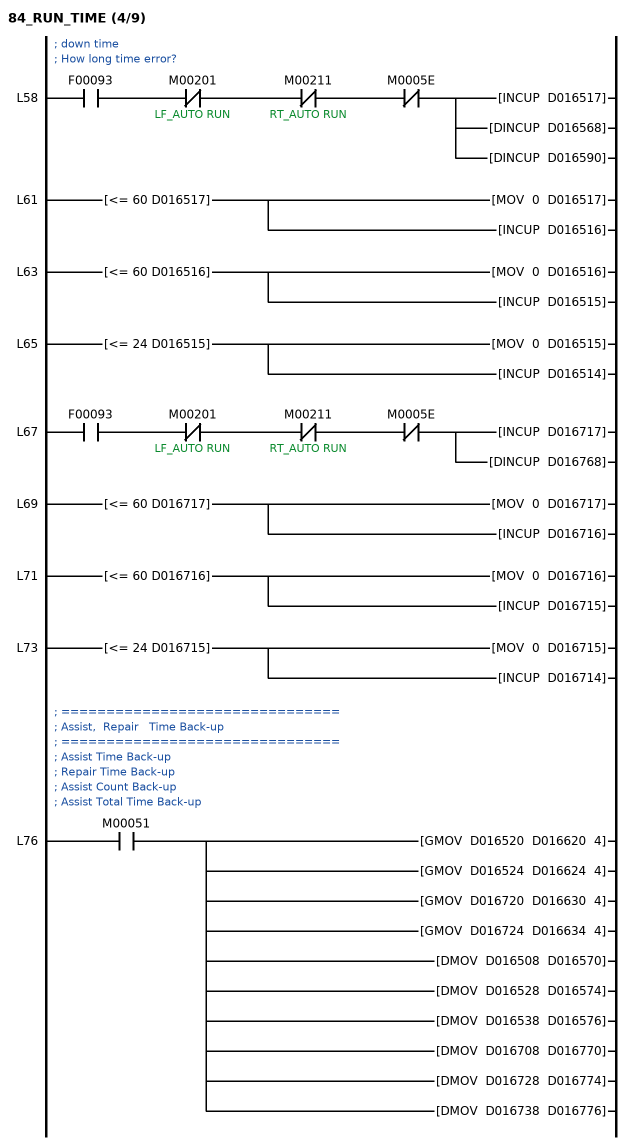
[picture p360: 84_RUN_TIME rungs L58-L76]
; L58
LOAD      F00093
AND NOT   M00201	// LF_AUTO RUN
AND NOT   M00211	// RT_AUTO RUN
AND NOT   M0005E
INCUP     D016517
DINCUP    D016568
DINCUP    D016590
// output comment: down time
// output comment: How long time error?
; L61
LOAD<=    60 D016517
MOV       0 D016517
INCUP     D016516
; L63
LOAD<=    60 D016516
MOV       0 D016516
INCUP     D016515
; L65
LOAD<=    24 D016515
MOV       0 D016515
INCUP     D016514
; L67
LOAD      F00093
AND NOT   M00201	// LF_AUTO RUN
AND NOT   M00211	// RT_AUTO RUN
AND NOT   M0005E
INCUP     D016717
DINCUP    D016768
; L69
LOAD<=    60 D016717
MOV       0 D016717
INCUP     D016716
; L71
LOAD<=    60 D016716
MOV       0 D016716
INCUP     D016715
; L73
LOAD<=    24 D016715
MOV       0 D016715
INCUP     D016714
// ===============================
// Assist,  Repair   Time Back-up
// ===============================
; L76
LOAD      M00051
GMOV      D016520 D016620 4
GMOV      D016524 D016624 4
GMOV      D016720 D016630 4
GMOV      D016724 D016634 4
DMOV      D016508 D016570
DMOV      D016528 D016574
DMOV      D016538 D016576
DMOV      D016708 D016770
DMOV      D016728 D016774
DMOV      D016738 D016776
// output comment: Assist Time Back-up
// output comment: Repair Time Back-up
// output comment: Assist Count Back-up
// output comment: Assist Total Time Back-up

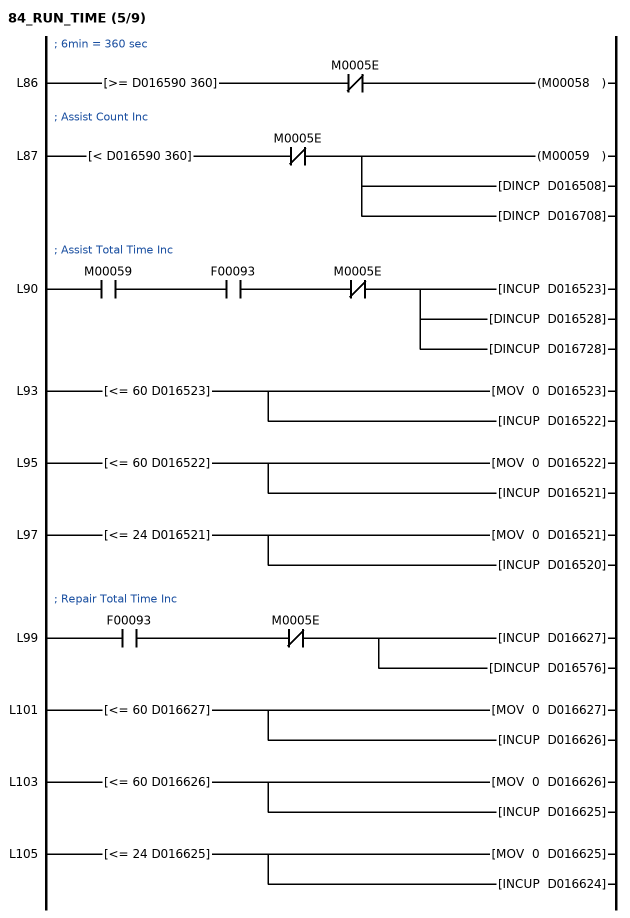
; L86
LOAD>=    D016590 360
AND NOT   M0005E
OUT       M00058
// output comment: 6min = 360 sec
; L87
LOAD<     D016590 360
AND NOT   M0005E
OUT       M00059
DINCP     D016508
DINCP     D016708
// output comment: Assist Count Inc
; L90
LOAD      M00059
AND       F00093
AND NOT   M0005E
INCUP     D016523
DINCUP    D016528
DINCUP    D016728
// output comment: Assist Total Time Inc
; L93
LOAD<=    60 D016523
MOV       0 D016523
INCUP     D016522
; L95
LOAD<=    60 D016522
MOV       0 D016522
INCUP     D016521
; L97
LOAD<=    24 D016521
MOV       0 D016521
INCUP     D016520
; L99
LOAD      F00093
AND NOT   M0005E
INCUP     D016627
DINCUP    D016576
// output comment: Repair Total Time Inc
; L101
LOAD<=    60 D016627
MOV       0 D016627
INCUP     D016626
; L103
LOAD<=    60 D016626
MOV       0 D016626
INCUP     D016625
; L105
LOAD<=    24 D016625
MOV       0 D016625
INCUP     D016624

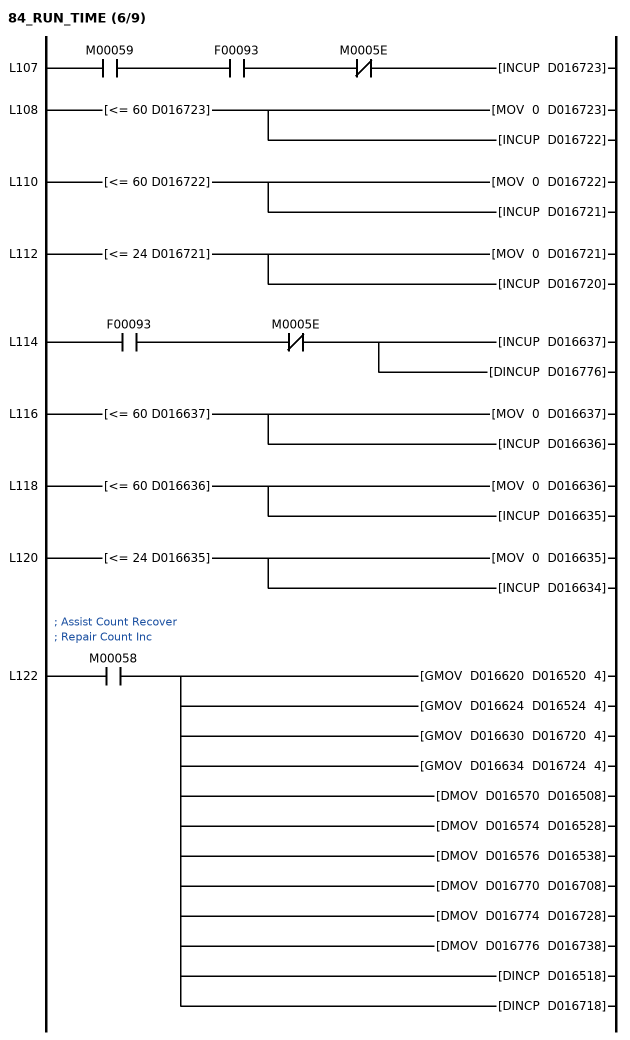
; L107
LOAD      M00059
AND       F00093
AND NOT   M0005E
INCUP     D016723
; L108
LOAD<=    60 D016723
MOV       0 D016723
INCUP     D016722
; L110
LOAD<=    60 D016722
MOV       0 D016722
INCUP     D016721
; L112
LOAD<=    24 D016721
MOV       0 D016721
INCUP     D016720
; L114
LOAD      F00093
AND NOT   M0005E
INCUP     D016637
DINCUP    D016776
; L116
LOAD<=    60 D016637
MOV       0 D016637
INCUP     D016636
; L118
LOAD<=    60 D016636
MOV       0 D016636
INCUP     D016635
; L120
LOAD<=    24 D016635
MOV       0 D016635
INCUP     D016634
; L122
LOAD      M00058
GMOV      D016620 D016520 4
GMOV      D016624 D016524 4
GMOV      D016630 D016720 4
GMOV      D016634 D016724 4
DMOV      D016570 D016508
DMOV      D016574 D016528
DMOV      D016576 D016538
DMOV      D016770 D016708
DMOV      D016774 D016728
DMOV      D016776 D016738
DINCP     D016518
DINCP     D016718
// output comment: Assist Count Recover
// output comment: Repair Count Inc

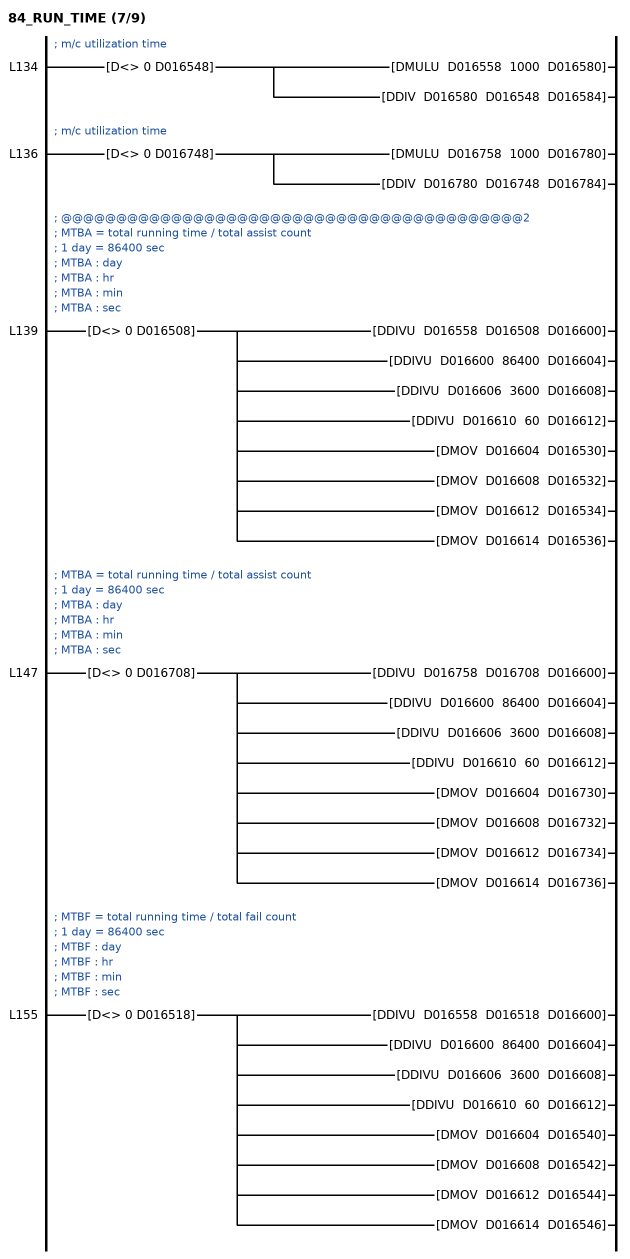
; L134
LOADD<>   0 D016548
DMULU     D016558 1000 D016580
DDIV      D016580 D016548 D016584
// output comment: m/c utilization time
; L136
LOADD<>   0 D016748
DMULU     D016758 1000 D016780
DDIV      D016780 D016748 D016784
// output comment: m/c utilization time
// @@@@@@@@@@@@@@@@@@@@@@@@@@@@@@@@@@@@@@@@@@2
; L139
LOADD<>   0 D016508
DDIVU     D016558 D016508 D016600
DDIVU     D016600 86400 D016604
DDIVU     D016606 3600 D016608
DDIVU     D016610 60 D016612
DMOV      D016604 D016530
DMOV      D016608 D016532
DMOV      D016612 D016534
DMOV      D016614 D016536
// output comment: MTBA = total running time / total assist count
// output comment: 1 day = 86400 sec
// output comment: MTBA : day
// output comment: MTBA : hr
// output comment: MTBA : min
// output comment: MTBA : sec
; L147
LOADD<>   0 D016708
DDIVU     D016758 D016708 D016600
DDIVU     D016600 86400 D016604
DDIVU     D016606 3600 D016608
DDIVU     D016610 60 D016612
DMOV      D016604 D016730
DMOV      D016608 D016732
DMOV      D016612 D016734
DMOV      D016614 D016736
// output comment: MTBA = total running time / total assist count
// output comment: 1 day = 86400 sec
// output comment: MTBA : day
// output comment: MTBA : hr
// output comment: MTBA : min
// output comment: MTBA : sec
; L155
LOADD<>   0 D016518
DDIVU     D016558 D016518 D016600
DDIVU     D016600 86400 D016604
DDIVU     D016606 3600 D016608
DDIVU     D016610 60 D016612
DMOV      D016604 D016540
DMOV      D016608 D016542
DMOV      D016612 D016544
DMOV      D016614 D016546
// output comment: MTBF = total running time / total fail count
// output comment: 1 day = 86400 sec
// output comment: MTBF : day
// output comment: MTBF : hr
// output comment: MTBF : min
// output comment: MTBF : sec

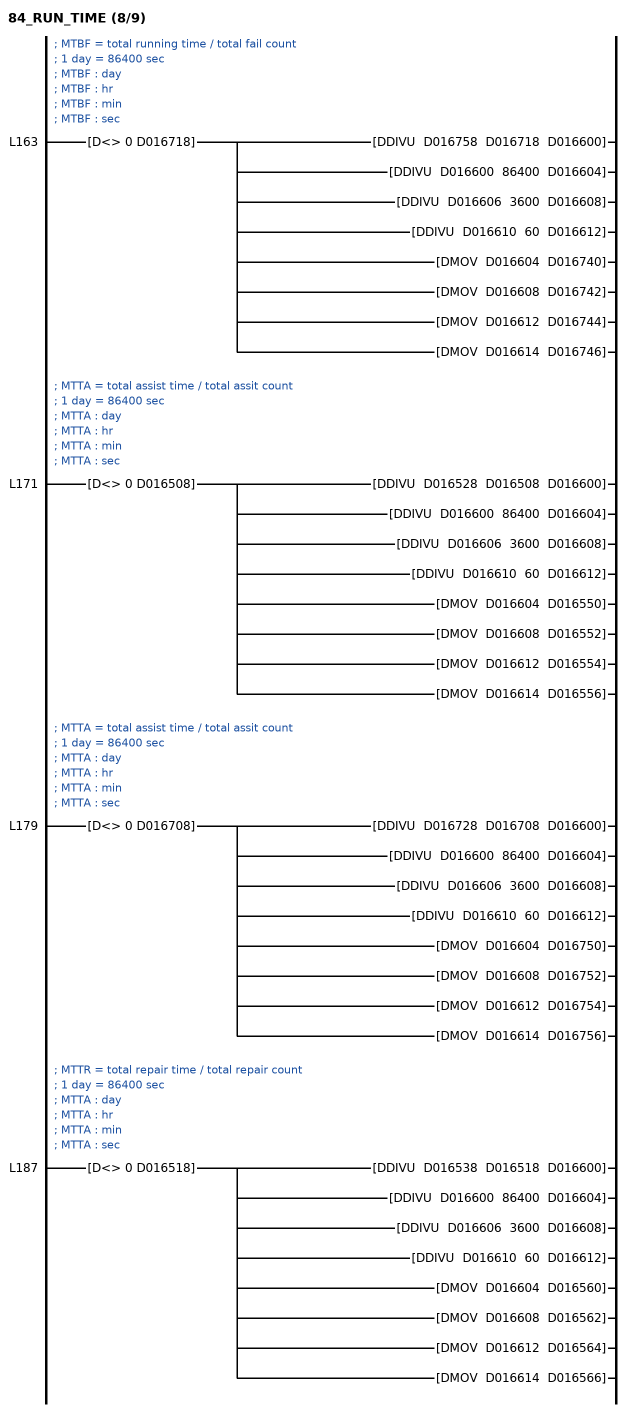
; L163
LOADD<>   0 D016718
DDIVU     D016758 D016718 D016600
DDIVU     D016600 86400 D016604
DDIVU     D016606 3600 D016608
DDIVU     D016610 60 D016612
DMOV      D016604 D016740
DMOV      D016608 D016742
DMOV      D016612 D016744
DMOV      D016614 D016746
// output comment: MTBF = total running time / total fail count
// output comment: 1 day = 86400 sec
// output comment: MTBF : day
// output comment: MTBF : hr
// output comment: MTBF : min
// output comment: MTBF : sec
; L171
LOADD<>   0 D016508
DDIVU     D016528 D016508 D016600
DDIVU     D016600 86400 D016604
DDIVU     D016606 3600 D016608
DDIVU     D016610 60 D016612
DMOV      D016604 D016550
DMOV      D016608 D016552
DMOV      D016612 D016554
DMOV      D016614 D016556
// output comment: MTTA = total assist time / total assit count
// output comment: 1 day = 86400 sec
// output comment: MTTA : day
// output comment: MTTA : hr
// output comment: MTTA : min
// output comment: MTTA : sec
; L179
LOADD<>   0 D016708
DDIVU     D016728 D016708 D016600
DDIVU     D016600 86400 D016604
DDIVU     D016606 3600 D016608
DDIVU     D016610 60 D016612
DMOV      D016604 D016750
DMOV      D016608 D016752
DMOV      D016612 D016754
DMOV      D016614 D016756
// output comment: MTTA = total assist time / total assit count
// output comment: 1 day = 86400 sec
// output comment: MTTA : day
// output comment: MTTA : hr
// output comment: MTTA : min
// output comment: MTTA : sec
; L187
LOADD<>   0 D016518
DDIVU     D016538 D016518 D016600
DDIVU     D016600 86400 D016604
DDIVU     D016606 3600 D016608
DDIVU     D016610 60 D016612
DMOV      D016604 D016560
DMOV      D016608 D016562
DMOV      D016612 D016564
DMOV      D016614 D016566
// output comment: MTTR = total repair time / total repair count
// output comment: 1 day = 86400 sec
// output comment: MTTA : day
// output comment: MTTA : hr
// output comment: MTTA : min
// output comment: MTTA : sec

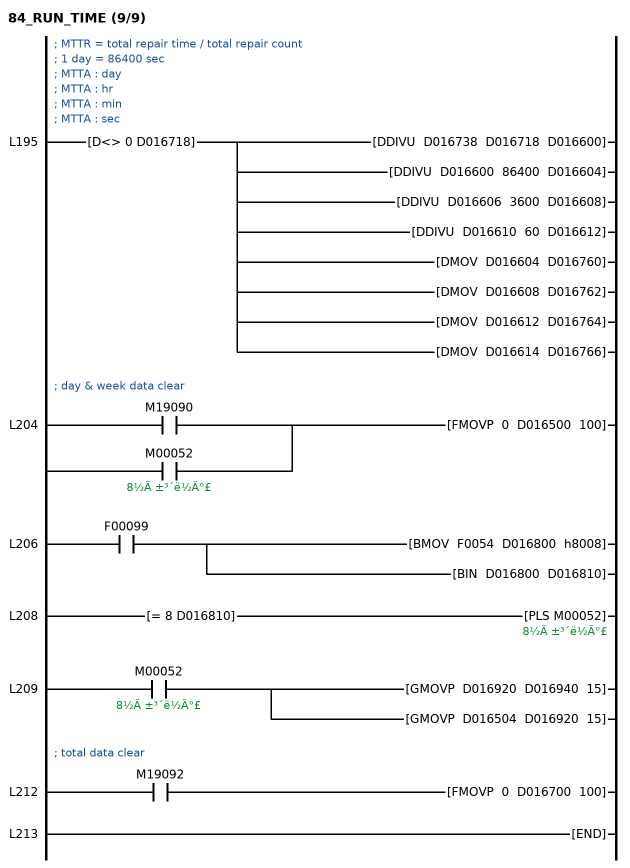
; L195
LOADD<>   0 D016718
DDIVU     D016738 D016718 D016600
DDIVU     D016600 86400 D016604
DDIVU     D016606 3600 D016608
DDIVU     D016610 60 D016612
DMOV      D016604 D016760
DMOV      D016608 D016762
DMOV      D016612 D016764
DMOV      D016614 D016766
// output comment: MTTR = total repair time / total repair count
// output comment: 1 day = 86400 sec
// output comment: MTTA : day
// output comment: MTTA : hr
// output comment: MTTA : min
// output comment: MTTA : sec
// day & week data clear
; L204
LOAD      M19090
OR        M00052	// 8½Ã ±³´ë½Ã°£
FMOVP     0 D016500 100
; L206
LOAD      F00099
BMOV      F0054 D016800 h8008
BIN       D016800 D016810
; L208
LOAD=     8 D016810
OUTP      M00052	// 8½Ã ±³´ë½Ã°£
; L209
LOAD      M00052	// 8½Ã ±³´ë½Ã°£
GMOVP     D016920 D016940 15
GMOVP     D016504 D016920 15
// total data clear
; L212
LOAD      M19092
FMOVP     0 D016700 100
; L213
END

PROGRAM 90_ALARM (task: ½ºÄµ ÇÁ·Î±×·¥)

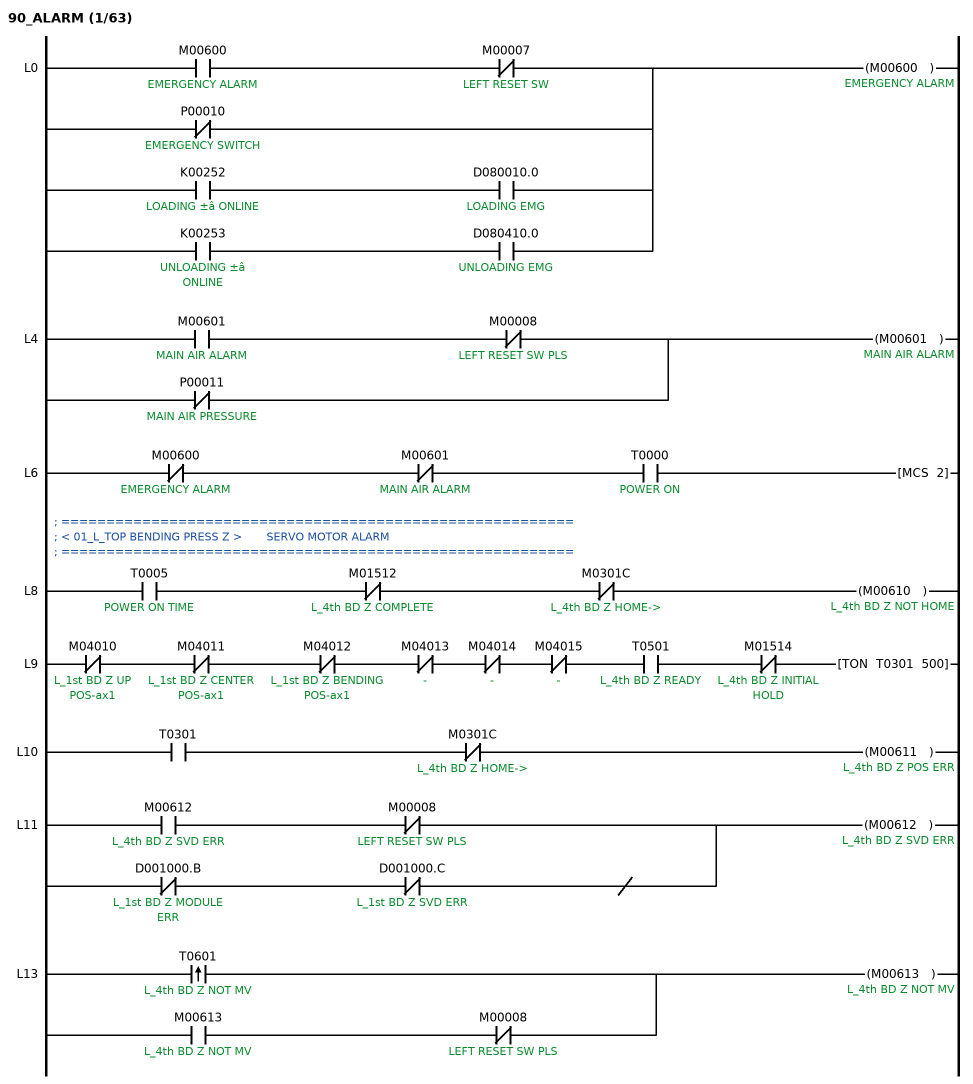
; L0
LOAD      M00600	// EMERGENCY ALARM
AND NOT   M00007	// LEFT RESET SW
OR NOT    P00010	// EMERGENCY SWITCH
LOAD      K00252	// LOADING ±â ONLINE
AND       D080010.0	// LOADING EMG
OR LOAD
LOAD      K00253	// UNLOADING ±â ONLINE
AND       D080410.0	// UNLOADING EMG
OR LOAD
OUT       M00600	// EMERGENCY ALARM
; L4
LOAD      M00601	// MAIN AIR ALARM
AND NOT   M00008	// LEFT RESET SW PLS
OR NOT    P00011	// MAIN AIR PRESSURE
OUT       M00601	// MAIN AIR ALARM
; L6
LOAD NOT  M00600	// EMERGENCY ALARM
AND NOT   M00601	// MAIN AIR ALARM
AND       T0000	// POWER ON
MCS       2
// =========================================================
// 
//        < 01_L_TOP BENDING PRESS Z >       SERVO MOTOR ALARM
// 
// =========================================================
; L8
LOAD      T0005	// POWER ON TIME
AND NOT   M01512	// L_4th BD Z COMPLETE
AND NOT   M0301C	// L_4th BD Z HOME->
OUT       M00610	// L_4th BD Z NOT HOME
; L9
LOAD NOT  M04010	// L_1st BD Z UP POS-ax1
AND NOT   M04011	// L_1st BD Z CENTER POS-ax1
AND NOT   M04012	// L_1st BD Z BENDING POS-ax1
AND NOT   M04013	// -
AND NOT   M04014	// -
AND NOT   M04015	// -
AND       T0501	// L_4th BD Z READY
AND NOT   M01514	// L_4th BD Z INITIAL HOLD
TON       T0301 500
; L10
LOAD      T0301
AND NOT   M0301C	// L_4th BD Z HOME->
OUT       M00611	// L_4th BD Z POS ERR
; L11
LOAD      M00612	// L_4th BD Z SVD ERR
AND NOT   M00008	// LEFT RESET SW PLS
LOAD NOT  D001000.B	// L_1st BD Z MODULE ERR
AND NOT   D001000.C	// L_1st BD Z SVD ERR
NOT
OR LOAD
OUT       M00612	// L_4th BD Z SVD ERR
; L13
LOADP     T0601	// L_4th BD Z NOT MV
LOAD      M00613	// L_4th BD Z NOT MV
AND NOT   M00008	// LEFT RESET SW PLS
OR LOAD
OUT       M00613	// L_4th BD Z NOT MV

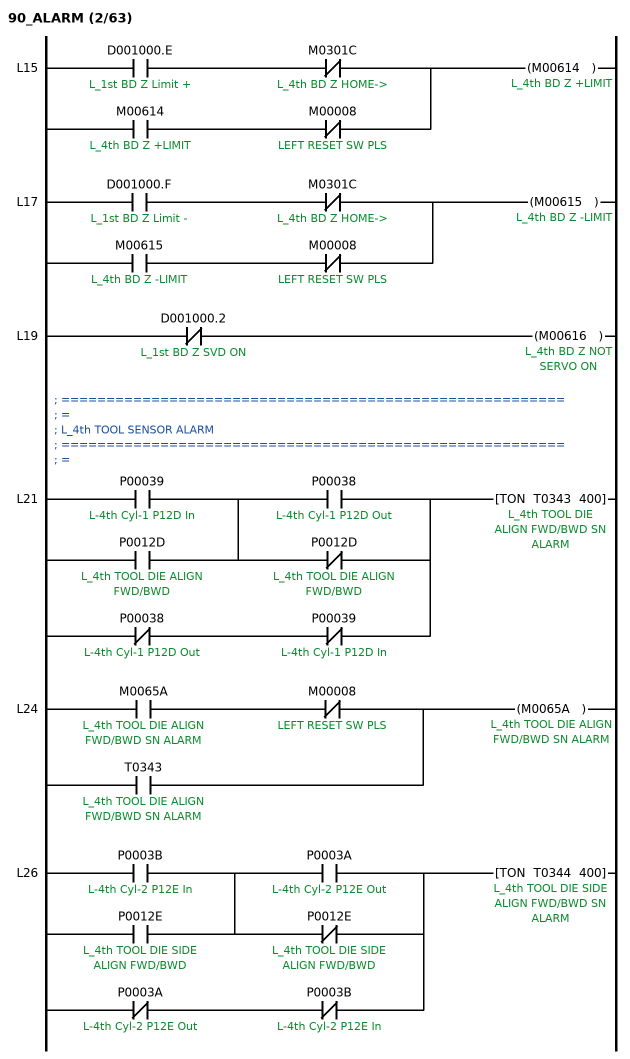
; L15
LOAD      D001000.E	// L_1st BD Z Limit +
AND NOT   M0301C	// L_4th BD Z HOME->
LOAD      M00614	// L_4th BD Z +LIMIT
AND NOT   M00008	// LEFT RESET SW PLS
OR LOAD
OUT       M00614	// L_4th BD Z +LIMIT
; L17
LOAD      D001000.F	// L_1st BD Z Limit -
AND NOT   M0301C	// L_4th BD Z HOME->
LOAD      M00615	// L_4th BD Z -LIMIT
AND NOT   M00008	// LEFT RESET SW PLS
OR LOAD
OUT       M00615	// L_4th BD Z -LIMIT
; L19
LOAD NOT  D001000.2	// L_1st BD Z SVD ON
OUT       M00616	// L_4th BD Z NOT SERVO ON
// =========================================================
// 
//        L_4th TOOL SENSOR ALARM
// 
// =========================================================
; L21
LOAD      P00039	// L-4th Cyl-1 P12D In
OR        P0012D	// L_4th TOOL DIE ALIGN FWD/BWD
LOAD      P00038	// L-4th Cyl-1 P12D Out
OR NOT    P0012D	// L_4th TOOL DIE ALIGN FWD/BWD
AND LOAD
LOAD NOT  P00038	// L-4th Cyl-1 P12D Out
AND NOT   P00039	// L-4th Cyl-1 P12D In
OR LOAD
TON       T0343 400	// L_4th TOOL DIE ALIGN FWD/BWD SN ALARM
; L24
LOAD      M0065A	// L_4th TOOL DIE ALIGN FWD/BWD SN ALARM
AND NOT   M00008	// LEFT RESET SW PLS
OR        T0343	// L_4th TOOL DIE ALIGN FWD/BWD SN ALARM
OUT       M0065A	// L_4th TOOL DIE ALIGN FWD/BWD SN ALARM
; L26
LOAD      P0003B	// L-4th Cyl-2 P12E In
OR        P0012E	// L_4th TOOL DIE SIDE ALIGN FWD/BWD
LOAD      P0003A	// L-4th Cyl-2 P12E Out
OR NOT    P0012E	// L_4th TOOL DIE SIDE ALIGN FWD/BWD
AND LOAD
LOAD NOT  P0003A	// L-4th Cyl-2 P12E Out
AND NOT   P0003B	// L-4th Cyl-2 P12E In
OR LOAD
TON       T0344 400	// L_4th TOOL DIE SIDE ALIGN FWD/BWD SN ALARM

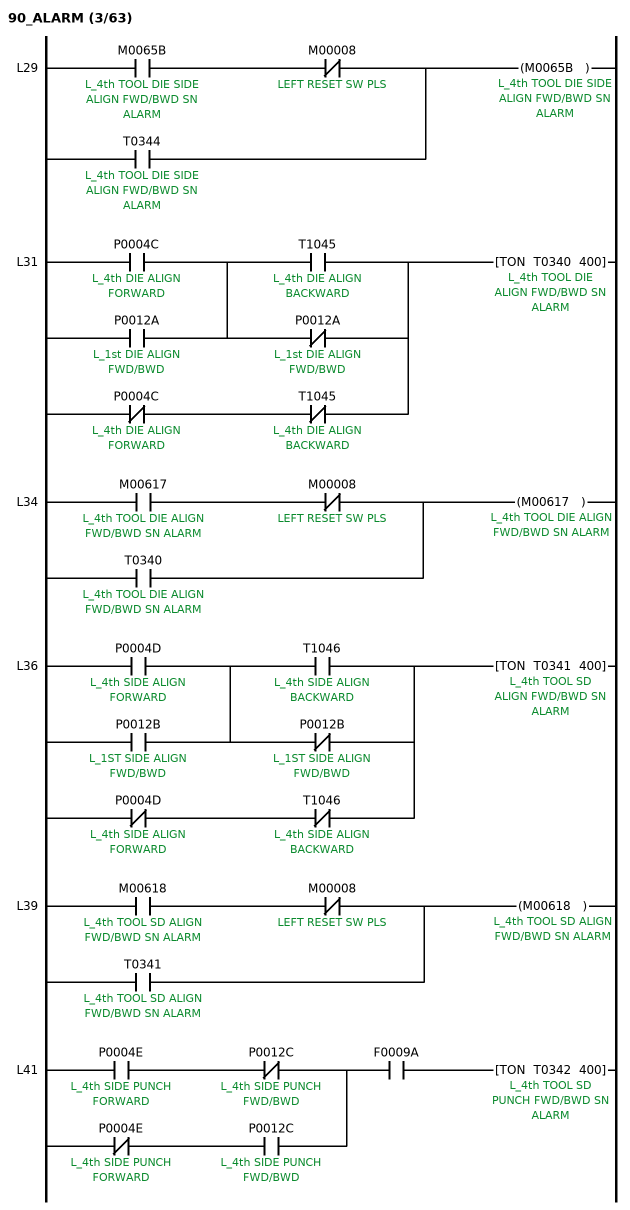
; L29
LOAD      M0065B	// L_4th TOOL DIE SIDE ALIGN FWD/BWD SN ALARM
AND NOT   M00008	// LEFT RESET SW PLS
OR        T0344	// L_4th TOOL DIE SIDE ALIGN FWD/BWD SN ALARM
OUT       M0065B	// L_4th TOOL DIE SIDE ALIGN FWD/BWD SN ALARM
; L31
LOAD      P0004C	// L_4th DIE ALIGN FORWARD
OR        P0012A	// L_1st DIE ALIGN FWD/BWD
LOAD      T1045	// L_4th DIE ALIGN BACKWARD
OR NOT    P0012A	// L_1st DIE ALIGN FWD/BWD
AND LOAD
LOAD NOT  P0004C	// L_4th DIE ALIGN FORWARD
AND NOT   T1045	// L_4th DIE ALIGN BACKWARD
OR LOAD
TON       T0340 400	// L_4th TOOL DIE ALIGN FWD/BWD SN ALARM
; L34
LOAD      M00617	// L_4th TOOL DIE ALIGN FWD/BWD SN ALARM
AND NOT   M00008	// LEFT RESET SW PLS
OR        T0340	// L_4th TOOL DIE ALIGN FWD/BWD SN ALARM
OUT       M00617	// L_4th TOOL DIE ALIGN FWD/BWD SN ALARM
; L36
LOAD      P0004D	// L_4th SIDE ALIGN FORWARD
OR        P0012B	// L_1ST SIDE ALIGN FWD/BWD
LOAD      T1046	// L_4th SIDE ALIGN BACKWARD
OR NOT    P0012B	// L_1ST SIDE ALIGN FWD/BWD
AND LOAD
LOAD NOT  P0004D	// L_4th SIDE ALIGN FORWARD
AND NOT   T1046	// L_4th SIDE ALIGN BACKWARD
OR LOAD
TON       T0341 400	// L_4th TOOL SD ALIGN FWD/BWD SN ALARM
; L39
LOAD      M00618	// L_4th TOOL SD ALIGN FWD/BWD SN ALARM
AND NOT   M00008	// LEFT RESET SW PLS
OR        T0341	// L_4th TOOL SD ALIGN FWD/BWD SN ALARM
OUT       M00618	// L_4th TOOL SD ALIGN FWD/BWD SN ALARM
; L41
LOAD      P0004E	// L_4th SIDE PUNCH FORWARD
AND NOT   P0012C	// L_4th SIDE PUNCH FWD/BWD
LOAD NOT  P0004E	// L_4th SIDE PUNCH FORWARD
AND       P0012C	// L_4th SIDE PUNCH FWD/BWD
OR LOAD
AND       F0009A
TON       T0342 400	// L_4th TOOL SD PUNCH FWD/BWD SN ALARM

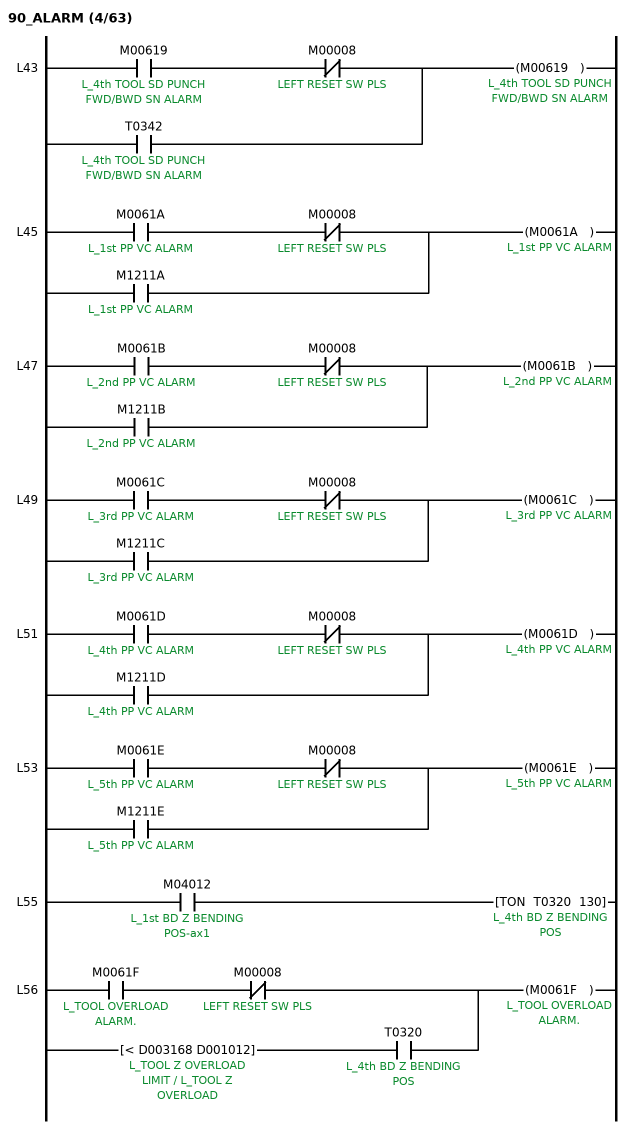
; L43
LOAD      M00619	// L_4th TOOL SD PUNCH FWD/BWD SN ALARM
AND NOT   M00008	// LEFT RESET SW PLS
OR        T0342	// L_4th TOOL SD PUNCH FWD/BWD SN ALARM
OUT       M00619	// L_4th TOOL SD PUNCH FWD/BWD SN ALARM
; L45
LOAD      M0061A	// L_1st PP VC ALARM
AND NOT   M00008	// LEFT RESET SW PLS
OR        M1211A	// L_1st PP VC ALARM
OUT       M0061A	// L_1st PP VC ALARM
; L47
LOAD      M0061B	// L_2nd PP VC ALARM
AND NOT   M00008	// LEFT RESET SW PLS
OR        M1211B	// L_2nd PP VC ALARM
OUT       M0061B	// L_2nd PP VC ALARM
; L49
LOAD      M0061C	// L_3rd PP VC ALARM
AND NOT   M00008	// LEFT RESET SW PLS
OR        M1211C	// L_3rd PP VC ALARM
OUT       M0061C	// L_3rd PP VC ALARM
; L51
LOAD      M0061D	// L_4th PP VC ALARM
AND NOT   M00008	// LEFT RESET SW PLS
OR        M1211D	// L_4th PP VC ALARM
OUT       M0061D	// L_4th PP VC ALARM
; L53
LOAD      M0061E	// L_5th PP VC ALARM
AND NOT   M00008	// LEFT RESET SW PLS
OR        M1211E	// L_5th PP VC ALARM
OUT       M0061E	// L_5th PP VC ALARM
; L55
LOAD      M04012	// L_1st BD Z BENDING POS-ax1
TON       T0320 130	// L_4th BD Z BENDING POS
; L56
LOAD      M0061F	// L_TOOL OVERLOAD ALARM.
AND NOT   M00008	// LEFT RESET SW PLS
LOAD<     D003168 D001012	// L_TOOL Z OVERLOAD LIMIT / L_TOOL Z OVERLOAD
AND       T0320	// L_4th BD Z BENDING POS
OR LOAD
OUT       M0061F	// L_TOOL OVERLOAD ALARM.

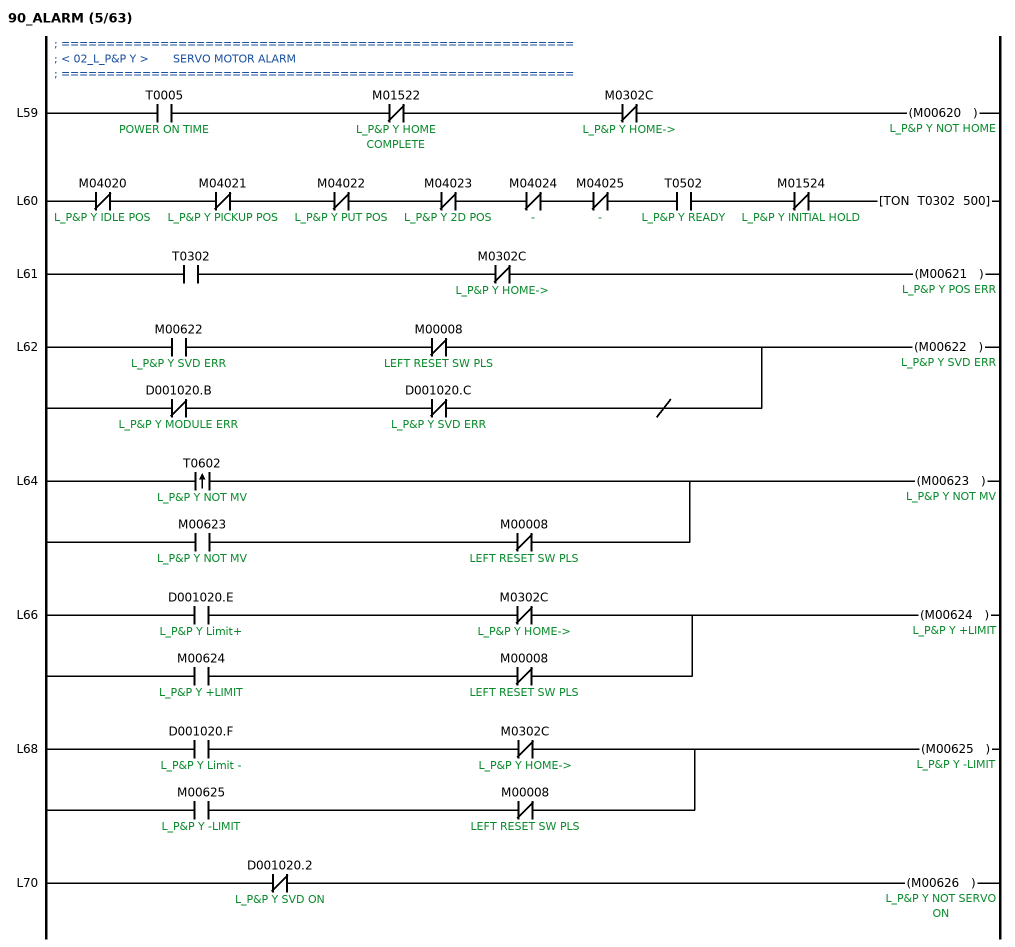
// =========================================================
// 
//        < 02_L_P&P Y >       SERVO MOTOR ALARM
// 
// =========================================================
; L59
LOAD      T0005	// POWER ON TIME
AND NOT   M01522	// L_P&P Y HOME COMPLETE
AND NOT   M0302C	// L_P&P Y HOME->
OUT       M00620	// L_P&P Y NOT HOME
; L60
LOAD NOT  M04020	// L_P&P Y IDLE POS
AND NOT   M04021	// L_P&P Y PICKUP POS
AND NOT   M04022	// L_P&P Y PUT POS
AND NOT   M04023	// L_P&P Y 2D POS
AND NOT   M04024	// -
AND NOT   M04025	// -
AND       T0502	// L_P&P Y READY
AND NOT   M01524	// L_P&P Y INITIAL HOLD
TON       T0302 500
; L61
LOAD      T0302
AND NOT   M0302C	// L_P&P Y HOME->
OUT       M00621	// L_P&P Y POS ERR
; L62
LOAD      M00622	// L_P&P Y SVD ERR
AND NOT   M00008	// LEFT RESET SW PLS
LOAD NOT  D001020.B	// L_P&P Y MODULE ERR
AND NOT   D001020.C	// L_P&P Y SVD ERR
NOT
OR LOAD
OUT       M00622	// L_P&P Y SVD ERR
; L64
LOADP     T0602	// L_P&P Y NOT MV
LOAD      M00623	// L_P&P Y NOT MV
AND NOT   M00008	// LEFT RESET SW PLS
OR LOAD
OUT       M00623	// L_P&P Y NOT MV
; L66
LOAD      D001020.E	// L_P&P Y Limit+
AND NOT   M0302C	// L_P&P Y HOME->
LOAD      M00624	// L_P&P Y +LIMIT
AND NOT   M00008	// LEFT RESET SW PLS
OR LOAD
OUT       M00624	// L_P&P Y +LIMIT
; L68
LOAD      D001020.F	// L_P&P Y Limit -
AND NOT   M0302C	// L_P&P Y HOME->
LOAD      M00625	// L_P&P Y -LIMIT
AND NOT   M00008	// LEFT RESET SW PLS
OR LOAD
OUT       M00625	// L_P&P Y -LIMIT
; L70
LOAD NOT  D001020.2	// L_P&P Y SVD ON
OUT       M00626	// L_P&P Y NOT SERVO ON

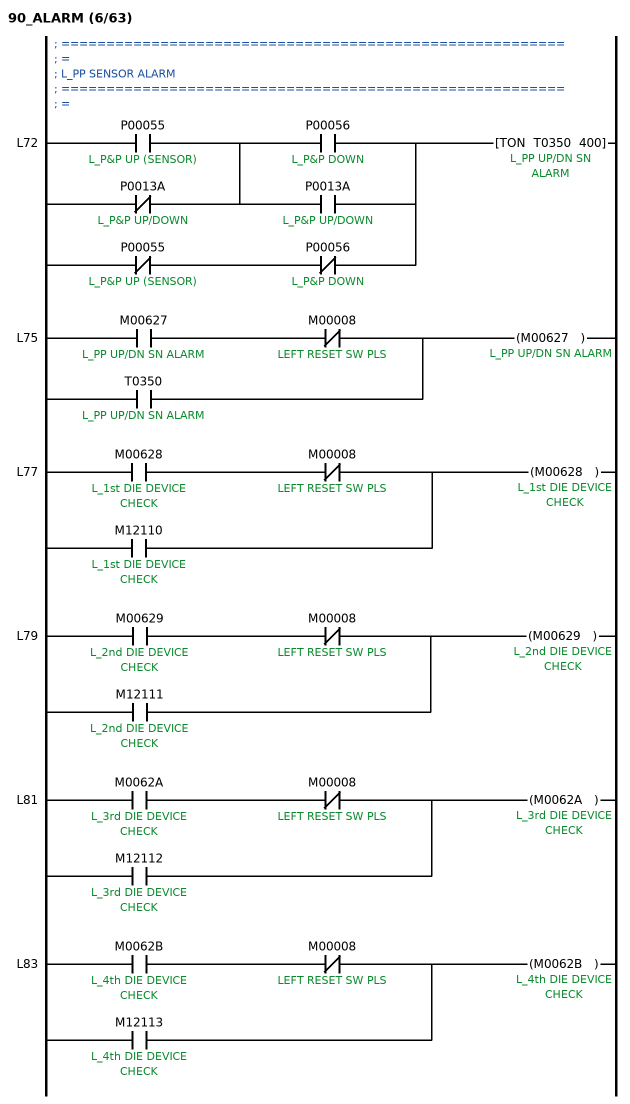
// =========================================================
// 
//       L_PP SENSOR ALARM
// 
// =========================================================
; L72
LOAD      P00055	// L_P&P UP (SENSOR)
OR NOT    P0013A	// L_P&P UP/DOWN
LOAD      P00056	// L_P&P DOWN
OR        P0013A	// L_P&P UP/DOWN
AND LOAD
LOAD NOT  P00055	// L_P&P UP (SENSOR)
AND NOT   P00056	// L_P&P DOWN
OR LOAD
TON       T0350 400	// L_PP UP/DN SN ALARM
; L75
LOAD      M00627	// L_PP UP/DN SN ALARM
AND NOT   M00008	// LEFT RESET SW PLS
OR        T0350	// L_PP UP/DN SN ALARM
OUT       M00627	// L_PP UP/DN SN ALARM
; L77
LOAD      M00628	// L_1st DIE DEVICE CHECK
AND NOT   M00008	// LEFT RESET SW PLS
OR        M12110	// L_1st DIE DEVICE CHECK
OUT       M00628	// L_1st DIE DEVICE CHECK
; L79
LOAD      M00629	// L_2nd DIE DEVICE CHECK
AND NOT   M00008	// LEFT RESET SW PLS
OR        M12111	// L_2nd DIE DEVICE CHECK
OUT       M00629	// L_2nd DIE DEVICE CHECK
; L81
LOAD      M0062A	// L_3rd DIE DEVICE CHECK
AND NOT   M00008	// LEFT RESET SW PLS
OR        M12112	// L_3rd DIE DEVICE CHECK
OUT       M0062A	// L_3rd DIE DEVICE CHECK
; L83
LOAD      M0062B	// L_4th DIE DEVICE CHECK
AND NOT   M00008	// LEFT RESET SW PLS
OR        M12113	// L_4th DIE DEVICE CHECK
OUT       M0062B	// L_4th DIE DEVICE CHECK

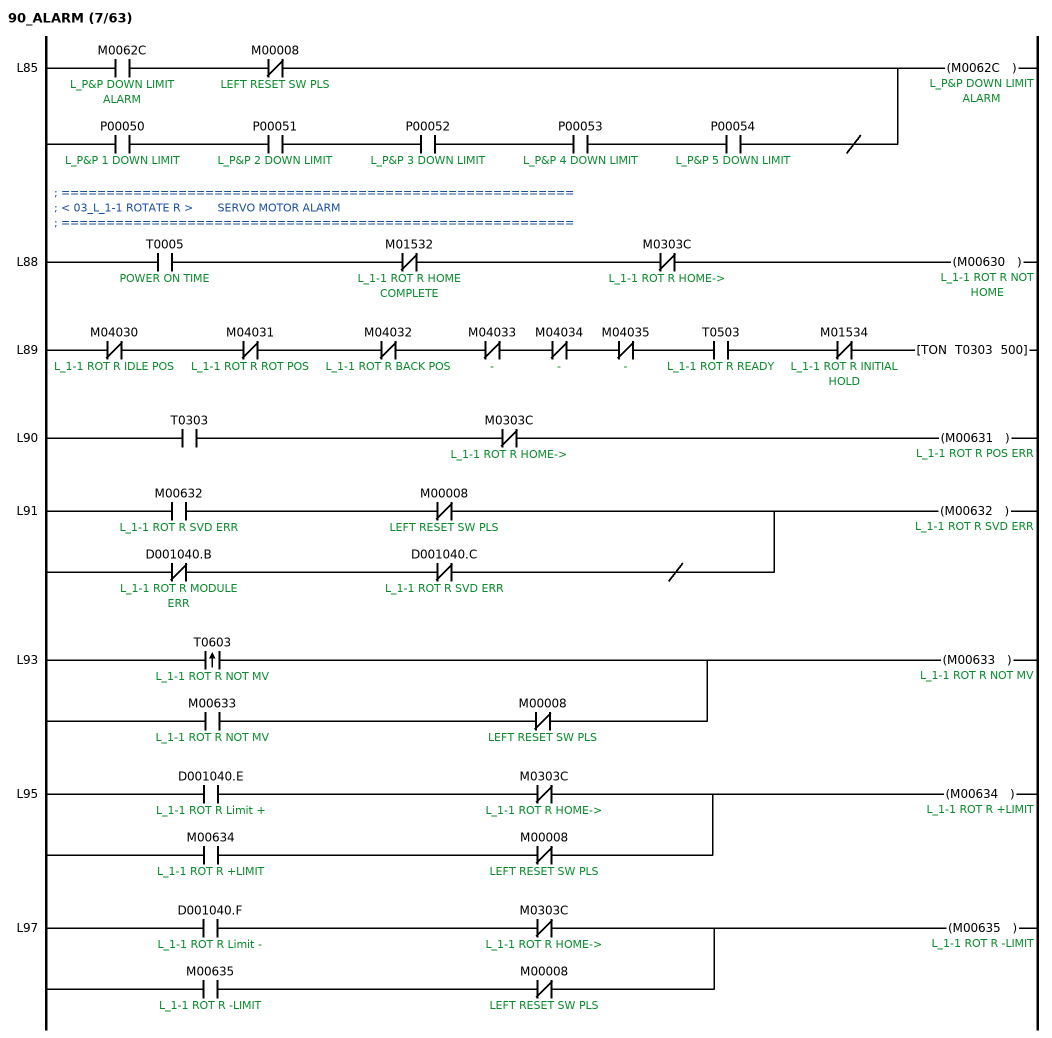
; L85
LOAD      M0062C	// L_P&P DOWN LIMIT ALARM
AND NOT   M00008	// LEFT RESET SW PLS
LOAD      P00050	// L_P&P 1 DOWN LIMIT
AND       P00051	// L_P&P 2 DOWN LIMIT
AND       P00052	// L_P&P 3 DOWN LIMIT
AND       P00053	// L_P&P 4 DOWN LIMIT
AND       P00054	// L_P&P 5 DOWN LIMIT
NOT
OR LOAD
OUT       M0062C	// L_P&P DOWN LIMIT ALARM
// =========================================================
// 
//        < 03_L_1-1 ROTATE R >       SERVO MOTOR ALARM
// 
// =========================================================
; L88
LOAD      T0005	// POWER ON TIME
AND NOT   M01532	// L_1-1 ROT R HOME COMPLETE
AND NOT   M0303C	// L_1-1 ROT R HOME->
OUT       M00630	// L_1-1 ROT R NOT HOME
; L89
LOAD NOT  M04030	// L_1-1 ROT R IDLE POS
AND NOT   M04031	// L_1-1 ROT R ROT POS
AND NOT   M04032	// L_1-1 ROT R BACK POS
AND NOT   M04033	// -
AND NOT   M04034	// -
AND NOT   M04035	// -
AND       T0503	// L_1-1 ROT R READY
AND NOT   M01534	// L_1-1 ROT R INITIAL HOLD
TON       T0303 500
; L90
LOAD      T0303
AND NOT   M0303C	// L_1-1 ROT R HOME->
OUT       M00631	// L_1-1 ROT R POS ERR
; L91
LOAD      M00632	// L_1-1 ROT R SVD ERR
AND NOT   M00008	// LEFT RESET SW PLS
LOAD NOT  D001040.B	// L_1-1 ROT R MODULE ERR
AND NOT   D001040.C	// L_1-1 ROT R SVD ERR
NOT
OR LOAD
OUT       M00632	// L_1-1 ROT R SVD ERR
; L93
LOADP     T0603	// L_1-1 ROT R NOT MV
LOAD      M00633	// L_1-1 ROT R NOT MV
AND NOT   M00008	// LEFT RESET SW PLS
OR LOAD
OUT       M00633	// L_1-1 ROT R NOT MV
; L95
LOAD      D001040.E	// L_1-1 ROT R Limit +
AND NOT   M0303C	// L_1-1 ROT R HOME->
LOAD      M00634	// L_1-1 ROT R +LIMIT
AND NOT   M00008	// LEFT RESET SW PLS
OR LOAD
OUT       M00634	// L_1-1 ROT R +LIMIT
; L97
LOAD      D001040.F	// L_1-1 ROT R Limit -
AND NOT   M0303C	// L_1-1 ROT R HOME->
LOAD      M00635	// L_1-1 ROT R -LIMIT
AND NOT   M00008	// LEFT RESET SW PLS
OR LOAD
OUT       M00635	// L_1-1 ROT R -LIMIT

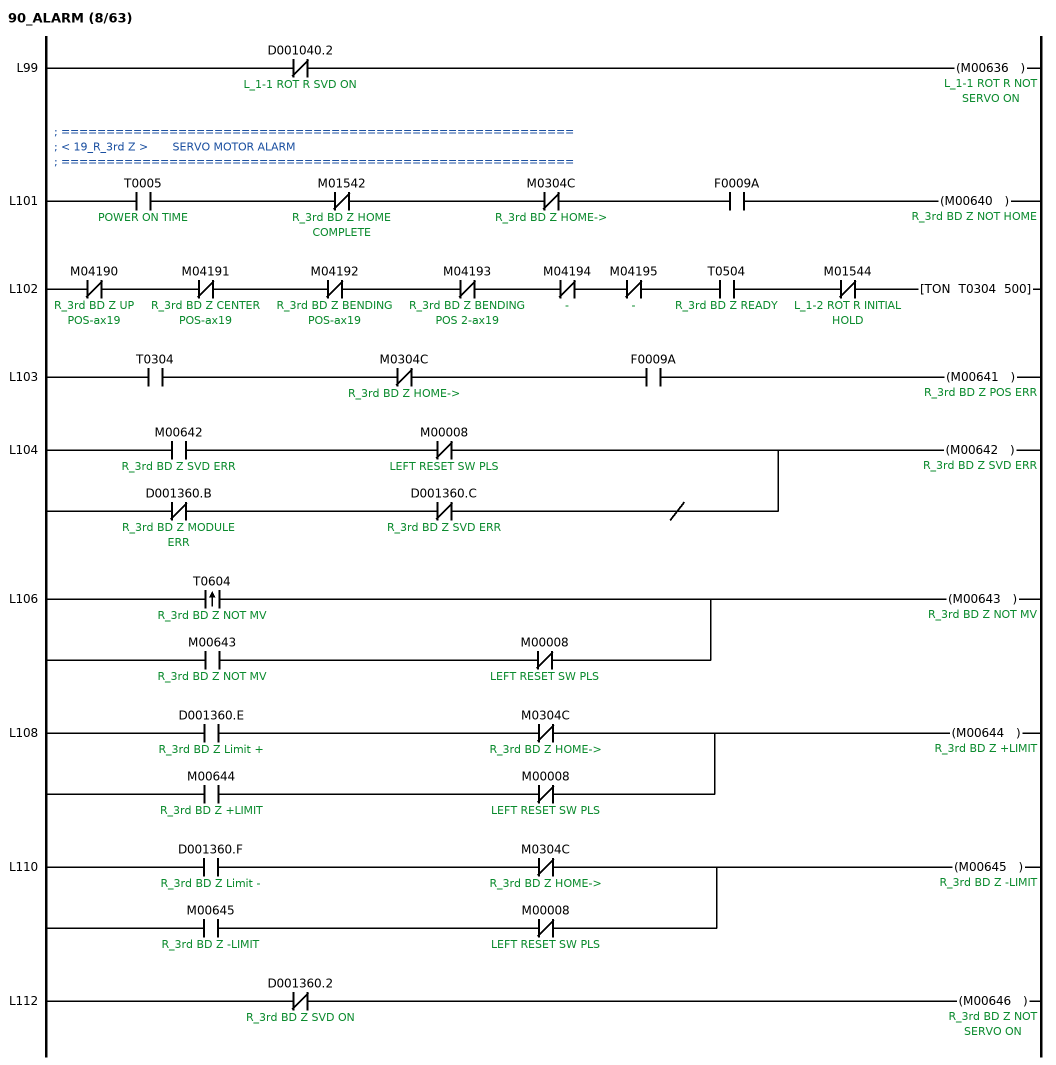
; L99
LOAD NOT  D001040.2	// L_1-1 ROT R SVD ON
OUT       M00636	// L_1-1 ROT R NOT SERVO ON
// =========================================================
// 
//        < 19_R_3rd Z >       SERVO MOTOR ALARM
// 
// =========================================================
; L101
LOAD      T0005	// POWER ON TIME
AND NOT   M01542	// R_3rd BD Z HOME COMPLETE
AND NOT   M0304C	// R_3rd BD Z HOME->
AND       F0009A
OUT       M00640	// R_3rd BD Z NOT HOME
; L102
LOAD NOT  M04190	// R_3rd BD Z UP POS-ax19
AND NOT   M04191	// R_3rd BD Z CENTER POS-ax19
AND NOT   M04192	// R_3rd BD Z BENDING POS-ax19
AND NOT   M04193	// R_3rd BD Z BENDING POS 2-ax19
AND NOT   M04194	// -
AND NOT   M04195	// -
AND       T0504	// R_3rd BD Z READY
AND NOT   M01544	// L_1-2 ROT R INITIAL HOLD
TON       T0304 500
; L103
LOAD      T0304
AND NOT   M0304C	// R_3rd BD Z HOME->
AND       F0009A
OUT       M00641	// R_3rd BD Z POS ERR
; L104
LOAD      M00642	// R_3rd BD Z SVD ERR
AND NOT   M00008	// LEFT RESET SW PLS
LOAD NOT  D001360.B	// R_3rd BD Z MODULE ERR
AND NOT   D001360.C	// R_3rd BD Z SVD ERR
NOT
OR LOAD
OUT       M00642	// R_3rd BD Z SVD ERR
; L106
LOADP     T0604	// R_3rd BD Z NOT MV
LOAD      M00643	// R_3rd BD Z NOT MV
AND NOT   M00008	// LEFT RESET SW PLS
OR LOAD
OUT       M00643	// R_3rd BD Z NOT MV
; L108
LOAD      D001360.E	// R_3rd BD Z Limit +
AND NOT   M0304C	// R_3rd BD Z HOME->
LOAD      M00644	// R_3rd BD Z +LIMIT
AND NOT   M00008	// LEFT RESET SW PLS
OR LOAD
OUT       M00644	// R_3rd BD Z +LIMIT
; L110
LOAD      D001360.F	// R_3rd BD Z Limit -
AND NOT   M0304C	// R_3rd BD Z HOME->
LOAD      M00645	// R_3rd BD Z -LIMIT
AND NOT   M00008	// LEFT RESET SW PLS
OR LOAD
OUT       M00645	// R_3rd BD Z -LIMIT
; L112
LOAD NOT  D001360.2	// R_3rd BD Z SVD ON
OUT       M00646	// R_3rd BD Z NOT SERVO ON

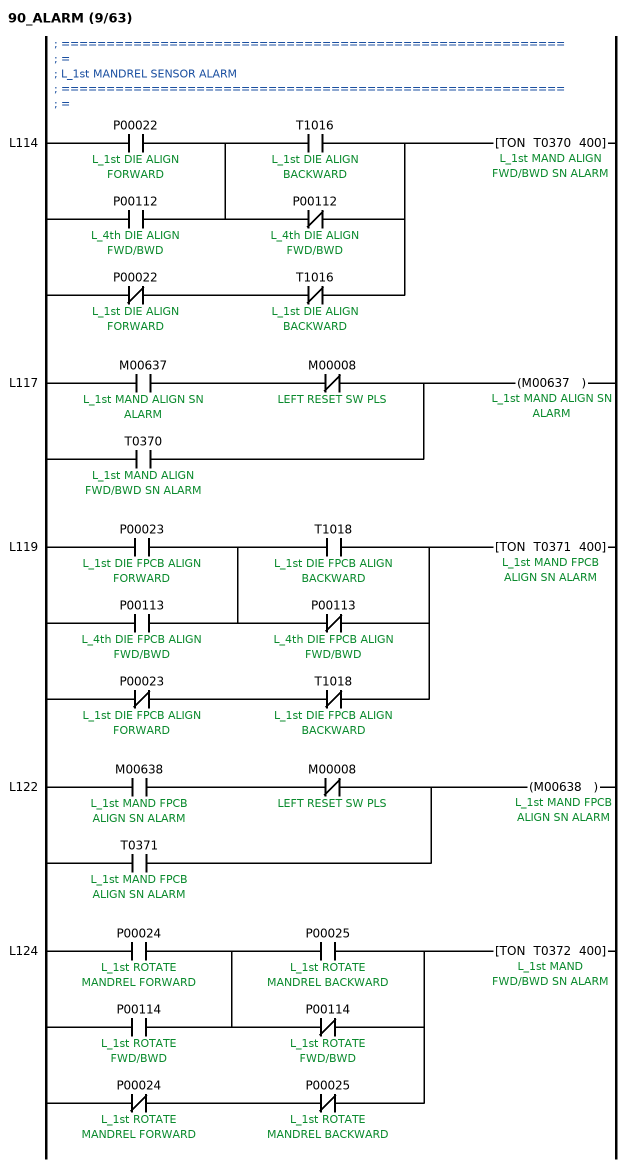
// =========================================================
// 
//        L_1st MANDREL SENSOR ALARM
// 
// =========================================================
; L114
LOAD      P00022	// L_1st DIE ALIGN FORWARD
OR        P00112	// L_4th DIE ALIGN FWD/BWD
LOAD      T1016	// L_1st DIE ALIGN BACKWARD
OR NOT    P00112	// L_4th DIE ALIGN FWD/BWD
AND LOAD
LOAD NOT  P00022	// L_1st DIE ALIGN FORWARD
AND NOT   T1016	// L_1st DIE ALIGN BACKWARD
OR LOAD
TON       T0370 400	// L_1st MAND ALIGN FWD/BWD SN ALARM
; L117
LOAD      M00637	// L_1st MAND ALIGN SN ALARM
AND NOT   M00008	// LEFT RESET SW PLS
OR        T0370	// L_1st MAND ALIGN FWD/BWD SN ALARM
OUT       M00637	// L_1st MAND ALIGN SN ALARM
; L119
LOAD      P00023	// L_1st DIE FPCB ALIGN FORWARD
OR        P00113	// L_4th DIE FPCB ALIGN FWD/BWD
LOAD      T1018	// L_1st DIE FPCB ALIGN BACKWARD
OR NOT    P00113	// L_4th DIE FPCB ALIGN FWD/BWD
AND LOAD
LOAD NOT  P00023	// L_1st DIE FPCB ALIGN FORWARD
AND NOT   T1018	// L_1st DIE FPCB ALIGN BACKWARD
OR LOAD
TON       T0371 400	// L_1st MAND FPCB ALIGN SN ALARM
; L122
LOAD      M00638	// L_1st MAND FPCB ALIGN SN ALARM
AND NOT   M00008	// LEFT RESET SW PLS
OR        T0371	// L_1st MAND FPCB ALIGN SN ALARM
OUT       M00638	// L_1st MAND FPCB ALIGN SN ALARM
; L124
LOAD      P00024	// L_1st ROTATE MANDREL FORWARD
OR        P00114	// L_1st ROTATE FWD/BWD
LOAD      P00025	// L_1st ROTATE MANDREL BACKWARD
OR NOT    P00114	// L_1st ROTATE FWD/BWD
AND LOAD
LOAD NOT  P00024	// L_1st ROTATE MANDREL FORWARD
AND NOT   P00025	// L_1st ROTATE MANDREL BACKWARD
OR LOAD
TON       T0372 400	// L_1st MAND FWD/BWD SN ALARM

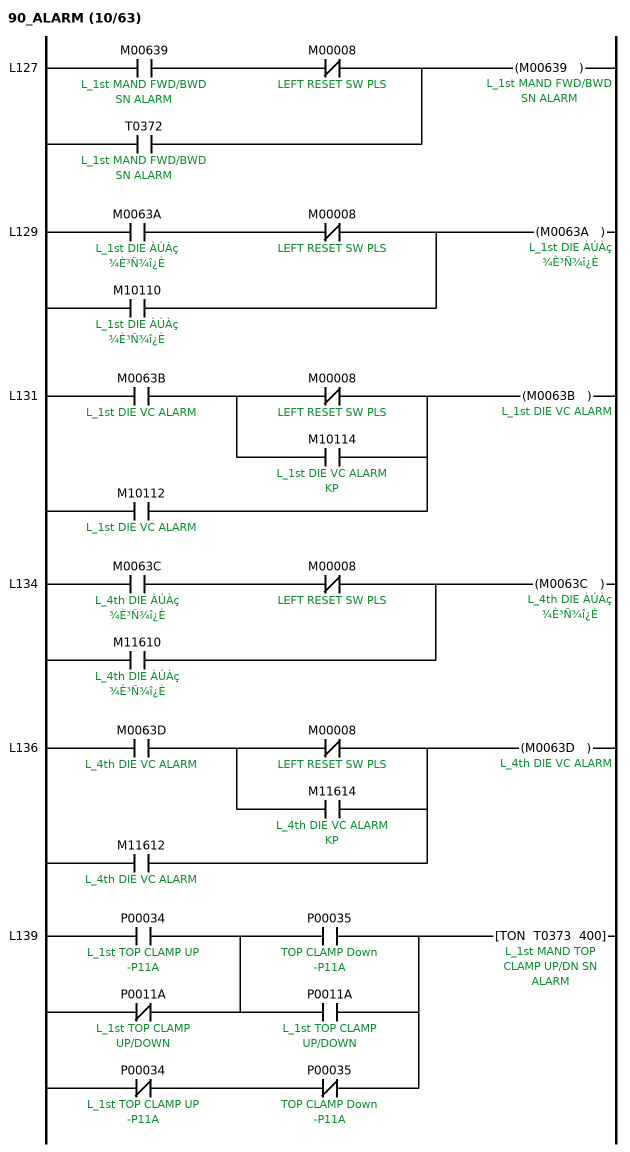
; L127
LOAD      M00639	// L_1st MAND FWD/BWD SN ALARM
AND NOT   M00008	// LEFT RESET SW PLS
OR        T0372	// L_1st MAND FWD/BWD SN ALARM
OUT       M00639	// L_1st MAND FWD/BWD SN ALARM
; L129
LOAD      M0063A	// L_1st DIE ÀÚÀç ¾È³Ñ¾î¿È
AND NOT   M00008	// LEFT RESET SW PLS
OR        M10110	// L_1st DIE ÀÚÀç ¾È³Ñ¾î¿È
OUT       M0063A	// L_1st DIE ÀÚÀç ¾È³Ñ¾î¿È
; L131
LOAD      M0063B	// L_1st DIE VC ALARM
LOAD NOT  M00008	// LEFT RESET SW PLS
OR        M10114	// L_1st DIE VC ALARM KP
AND LOAD
OR        M10112	// L_1st DIE VC ALARM
OUT       M0063B	// L_1st DIE VC ALARM
; L134
LOAD      M0063C	// L_4th DIE ÀÚÀç ¾È³Ñ¾î¿È
AND NOT   M00008	// LEFT RESET SW PLS
OR        M11610	// L_4th DIE ÀÚÀç ¾È³Ñ¾î¿È
OUT       M0063C	// L_4th DIE ÀÚÀç ¾È³Ñ¾î¿È
; L136
LOAD      M0063D	// L_4th DIE VC ALARM
LOAD NOT  M00008	// LEFT RESET SW PLS
OR        M11614	// L_4th DIE VC ALARM KP
AND LOAD
OR        M11612	// L_4th DIE VC ALARM
OUT       M0063D	// L_4th DIE VC ALARM
; L139
LOAD      P00034	// L_1st TOP CLAMP UP -P11A
OR NOT    P0011A	// L_1st TOP CLAMP UP/DOWN
LOAD      P00035	// TOP CLAMP Down -P11A
OR        P0011A	// L_1st TOP CLAMP UP/DOWN
AND LOAD
LOAD NOT  P00034	// L_1st TOP CLAMP UP -P11A
AND NOT   P00035	// TOP CLAMP Down -P11A
OR LOAD
TON       T0373 400	// L_1st MAND TOP CLAMP UP/DN SN ALARM

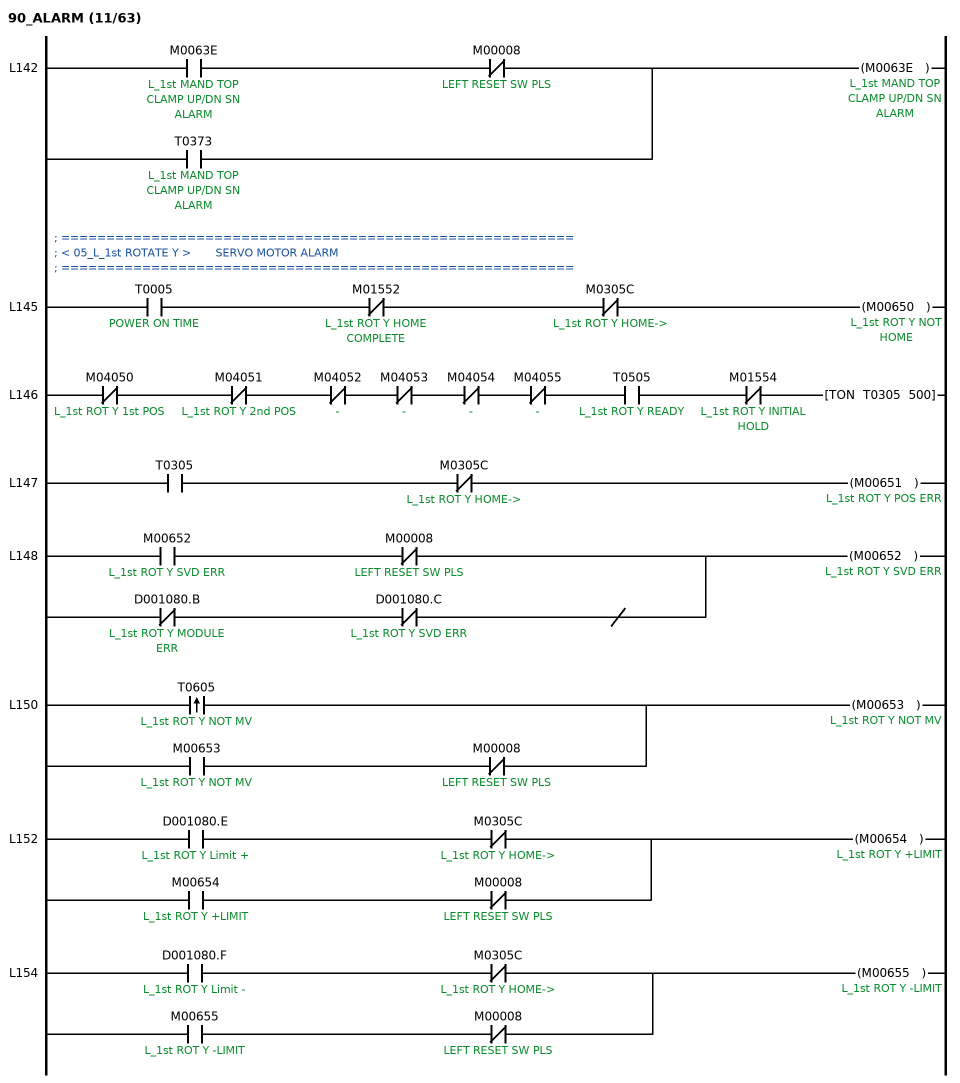
; L142
LOAD      M0063E	// L_1st MAND TOP CLAMP UP/DN SN ALARM
AND NOT   M00008	// LEFT RESET SW PLS
OR        T0373	// L_1st MAND TOP CLAMP UP/DN SN ALARM
OUT       M0063E	// L_1st MAND TOP CLAMP UP/DN SN ALARM
// =========================================================
// 
//        < 05_L_1st ROTATE Y >       SERVO MOTOR ALARM
// 
// =========================================================
; L145
LOAD      T0005	// POWER ON TIME
AND NOT   M01552	// L_1st ROT Y HOME COMPLETE
AND NOT   M0305C	// L_1st ROT Y HOME->
OUT       M00650	// L_1st ROT Y NOT HOME
; L146
LOAD NOT  M04050	// L_1st ROT Y 1st POS
AND NOT   M04051	// L_1st ROT Y 2nd POS
AND NOT   M04052	// -
AND NOT   M04053	// -
AND NOT   M04054	// -
AND NOT   M04055	// -
AND       T0505	// L_1st ROT Y READY
AND NOT   M01554	// L_1st ROT Y INITIAL HOLD
TON       T0305 500
; L147
LOAD      T0305
AND NOT   M0305C	// L_1st ROT Y HOME->
OUT       M00651	// L_1st ROT Y POS ERR
; L148
LOAD      M00652	// L_1st ROT Y SVD ERR
AND NOT   M00008	// LEFT RESET SW PLS
LOAD NOT  D001080.B	// L_1st ROT Y MODULE ERR
AND NOT   D001080.C	// L_1st ROT Y SVD ERR
NOT
OR LOAD
OUT       M00652	// L_1st ROT Y SVD ERR
; L150
LOADP     T0605	// L_1st ROT Y NOT MV
LOAD      M00653	// L_1st ROT Y NOT MV
AND NOT   M00008	// LEFT RESET SW PLS
OR LOAD
OUT       M00653	// L_1st ROT Y NOT MV
; L152
LOAD      D001080.E	// L_1st ROT Y Limit +
AND NOT   M0305C	// L_1st ROT Y HOME->
LOAD      M00654	// L_1st ROT Y +LIMIT
AND NOT   M00008	// LEFT RESET SW PLS
OR LOAD
OUT       M00654	// L_1st ROT Y +LIMIT
; L154
LOAD      D001080.F	// L_1st ROT Y Limit -
AND NOT   M0305C	// L_1st ROT Y HOME->
LOAD      M00655	// L_1st ROT Y -LIMIT
AND NOT   M00008	// LEFT RESET SW PLS
OR LOAD
OUT       M00655	// L_1st ROT Y -LIMIT

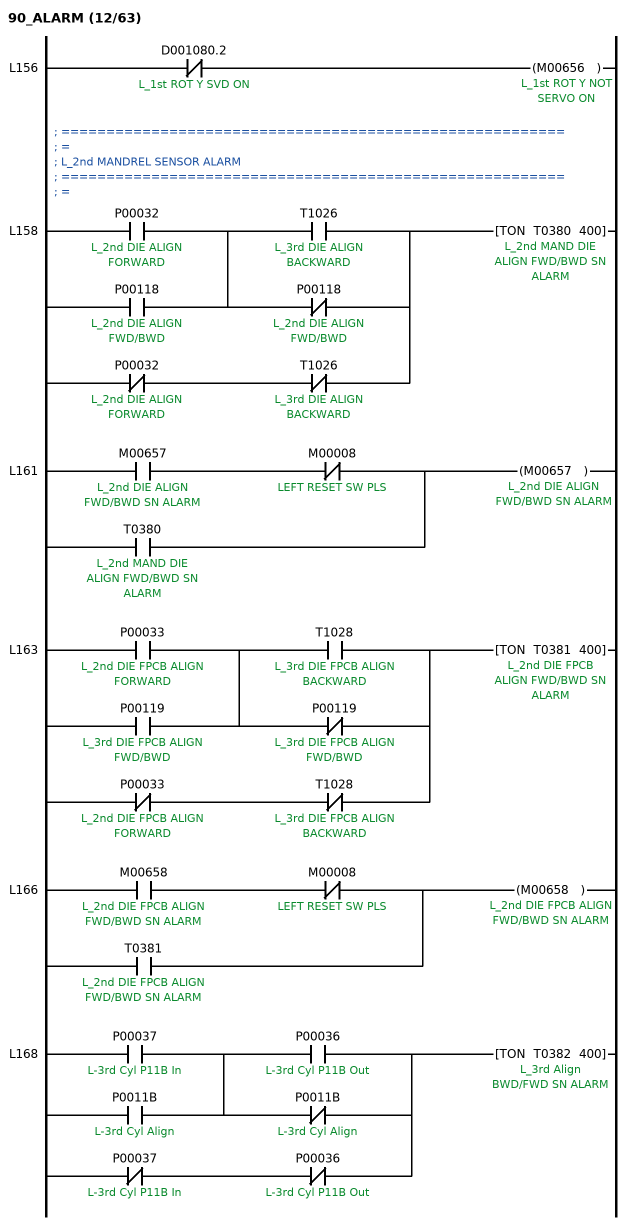
; L156
LOAD NOT  D001080.2	// L_1st ROT Y SVD ON
OUT       M00656	// L_1st ROT Y NOT SERVO ON
// =========================================================
// 
//        L_2nd MANDREL SENSOR ALARM
// 
// =========================================================
; L158
LOAD      P00032	// L_2nd DIE ALIGN FORWARD
OR        P00118	// L_2nd DIE ALIGN FWD/BWD
LOAD      T1026	// L_3rd DIE ALIGN BACKWARD
OR NOT    P00118	// L_2nd DIE ALIGN FWD/BWD
AND LOAD
LOAD NOT  P00032	// L_2nd DIE ALIGN FORWARD
AND NOT   T1026	// L_3rd DIE ALIGN BACKWARD
OR LOAD
TON       T0380 400	// L_2nd MAND DIE ALIGN FWD/BWD SN ALARM
; L161
LOAD      M00657	// L_2nd DIE ALIGN FWD/BWD SN ALARM
AND NOT   M00008	// LEFT RESET SW PLS
OR        T0380	// L_2nd MAND DIE ALIGN FWD/BWD SN ALARM
OUT       M00657	// L_2nd DIE ALIGN FWD/BWD SN ALARM
; L163
LOAD      P00033	// L_2nd DIE FPCB ALIGN FORWARD
OR        P00119	// L_3rd DIE FPCB ALIGN FWD/BWD
LOAD      T1028	// L_3rd DIE FPCB ALIGN BACKWARD
OR NOT    P00119	// L_3rd DIE FPCB ALIGN FWD/BWD
AND LOAD
LOAD NOT  P00033	// L_2nd DIE FPCB ALIGN FORWARD
AND NOT   T1028	// L_3rd DIE FPCB ALIGN BACKWARD
OR LOAD
TON       T0381 400	// L_2nd DIE FPCB ALIGN FWD/BWD SN ALARM
; L166
LOAD      M00658	// L_2nd DIE FPCB ALIGN FWD/BWD SN ALARM
AND NOT   M00008	// LEFT RESET SW PLS
OR        T0381	// L_2nd DIE FPCB ALIGN FWD/BWD SN ALARM
OUT       M00658	// L_2nd DIE FPCB ALIGN FWD/BWD SN ALARM
; L168
LOAD      P00037	// L-3rd Cyl P11B In
OR        P0011B	// L-3rd Cyl Align
LOAD      P00036	// L-3rd Cyl P11B Out
OR NOT    P0011B	// L-3rd Cyl Align
AND LOAD
LOAD NOT  P00037	// L-3rd Cyl P11B In
AND NOT   P00036	// L-3rd Cyl P11B Out
OR LOAD
TON       T0382 400	// L_3rd Align BWD/FWD SN ALARM

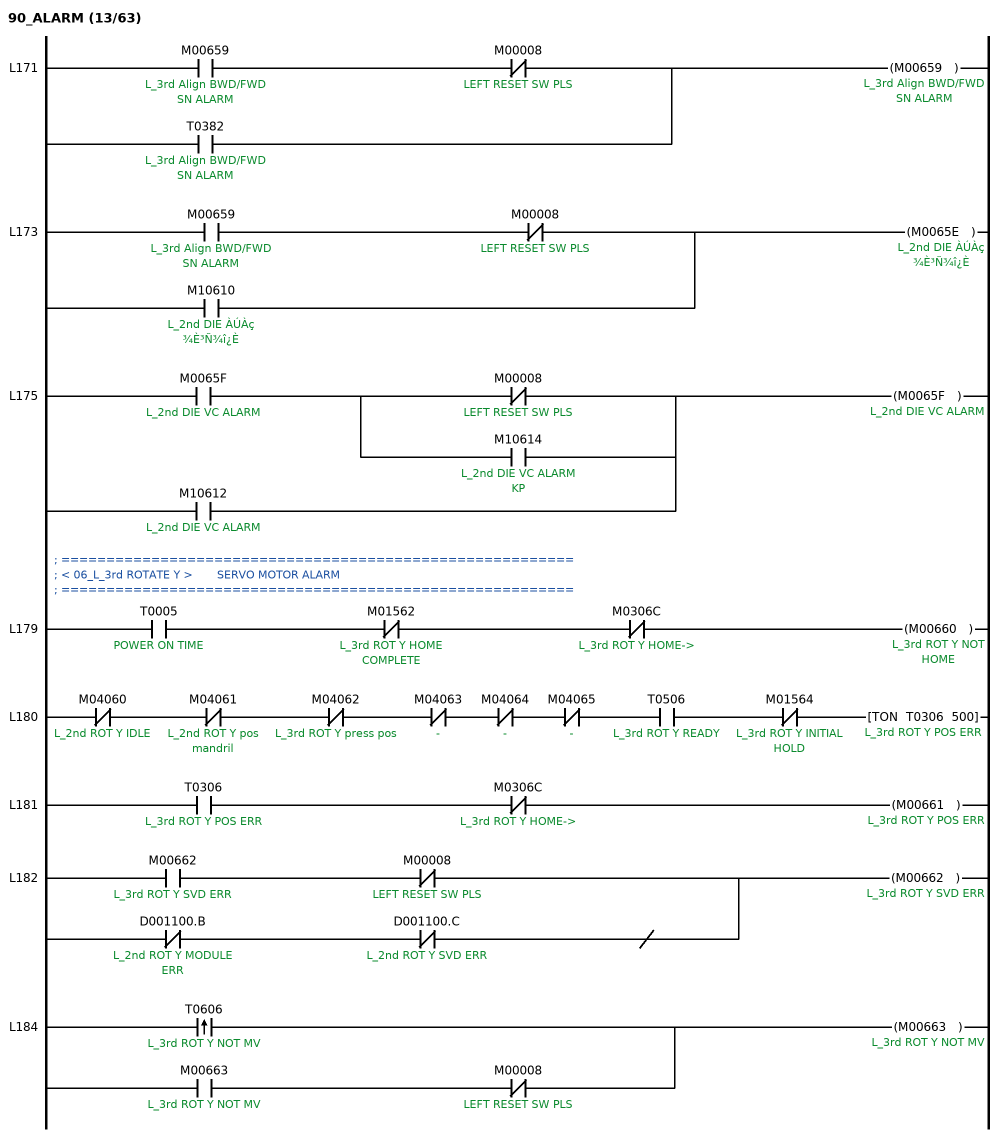
; L171
LOAD      M00659	// L_3rd Align BWD/FWD SN ALARM
AND NOT   M00008	// LEFT RESET SW PLS
OR        T0382	// L_3rd Align BWD/FWD SN ALARM
OUT       M00659	// L_3rd Align BWD/FWD SN ALARM
; L173
LOAD      M00659	// L_3rd Align BWD/FWD SN ALARM
AND NOT   M00008	// LEFT RESET SW PLS
OR        M10610	// L_2nd DIE ÀÚÀç ¾È³Ñ¾î¿È
OUT       M0065E	// L_2nd DIE ÀÚÀç ¾È³Ñ¾î¿È
; L175
LOAD      M0065F	// L_2nd DIE VC ALARM
LOAD NOT  M00008	// LEFT RESET SW PLS
OR        M10614	// L_2nd DIE VC ALARM KP
AND LOAD
OR        M10612	// L_2nd DIE VC ALARM
OUT       M0065F	// L_2nd DIE VC ALARM
// =========================================================
// 
//        < 06_L_3rd ROTATE Y >       SERVO MOTOR ALARM
// 
// =========================================================
; L179
LOAD      T0005	// POWER ON TIME
AND NOT   M01562	// L_3rd ROT Y HOME COMPLETE
AND NOT   M0306C	// L_3rd ROT Y HOME->
OUT       M00660	// L_3rd ROT Y NOT HOME
; L180
LOAD NOT  M04060	// L_2nd ROT Y IDLE
AND NOT   M04061	// L_2nd ROT Y pos mandril
AND NOT   M04062	// L_3rd ROT Y press pos
AND NOT   M04063	// -
AND NOT   M04064	// -
AND NOT   M04065	// -
AND       T0506	// L_3rd ROT Y READY
AND NOT   M01564	// L_3rd ROT Y INITIAL HOLD
TON       T0306 500	// L_3rd ROT Y POS ERR
; L181
LOAD      T0306	// L_3rd ROT Y POS ERR
AND NOT   M0306C	// L_3rd ROT Y HOME->
OUT       M00661	// L_3rd ROT Y POS ERR
; L182
LOAD      M00662	// L_3rd ROT Y SVD ERR
AND NOT   M00008	// LEFT RESET SW PLS
LOAD NOT  D001100.B	// L_2nd ROT Y MODULE ERR
AND NOT   D001100.C	// L_2nd ROT Y SVD ERR
NOT
OR LOAD
OUT       M00662	// L_3rd ROT Y SVD ERR
; L184
LOADP     T0606	// L_3rd ROT Y NOT MV
LOAD      M00663	// L_3rd ROT Y NOT MV
AND NOT   M00008	// LEFT RESET SW PLS
OR LOAD
OUT       M00663	// L_3rd ROT Y NOT MV

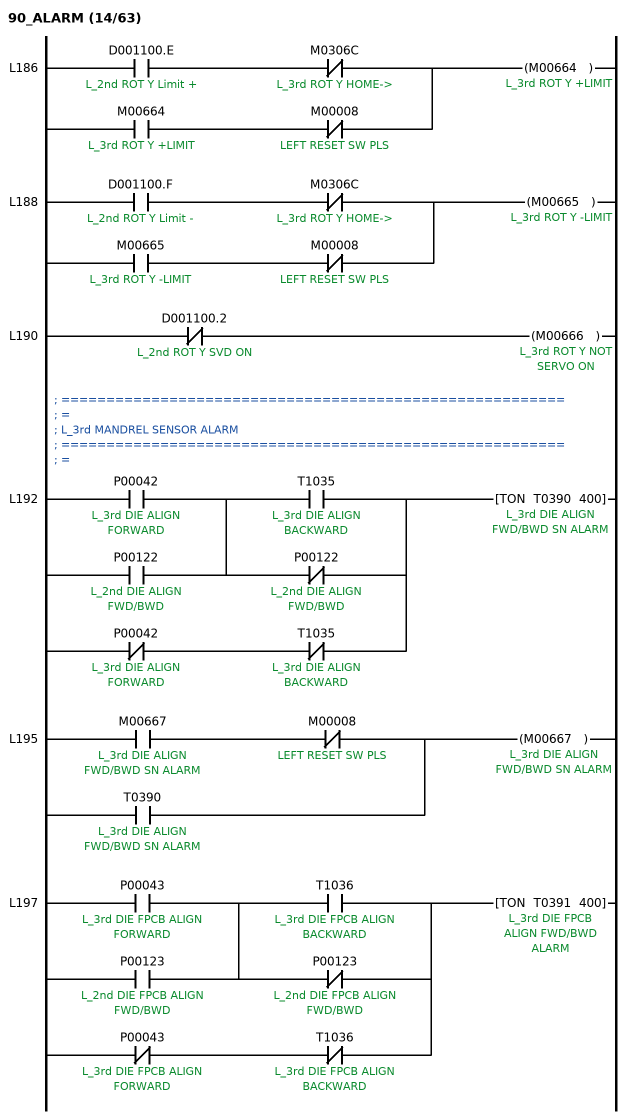
; L186
LOAD      D001100.E	// L_2nd ROT Y Limit +
AND NOT   M0306C	// L_3rd ROT Y HOME->
LOAD      M00664	// L_3rd ROT Y +LIMIT
AND NOT   M00008	// LEFT RESET SW PLS
OR LOAD
OUT       M00664	// L_3rd ROT Y +LIMIT
; L188
LOAD      D001100.F	// L_2nd ROT Y Limit -
AND NOT   M0306C	// L_3rd ROT Y HOME->
LOAD      M00665	// L_3rd ROT Y -LIMIT
AND NOT   M00008	// LEFT RESET SW PLS
OR LOAD
OUT       M00665	// L_3rd ROT Y -LIMIT
; L190
LOAD NOT  D001100.2	// L_2nd ROT Y SVD ON
OUT       M00666	// L_3rd ROT Y NOT SERVO ON
// =========================================================
// 
//        L_3rd MANDREL SENSOR ALARM
// 
// =========================================================
; L192
LOAD      P00042	// L_3rd DIE ALIGN FORWARD
OR        P00122	// L_2nd DIE ALIGN FWD/BWD
LOAD      T1035	// L_3rd DIE ALIGN BACKWARD
OR NOT    P00122	// L_2nd DIE ALIGN FWD/BWD
AND LOAD
LOAD NOT  P00042	// L_3rd DIE ALIGN FORWARD
AND NOT   T1035	// L_3rd DIE ALIGN BACKWARD
OR LOAD
TON       T0390 400	// L_3rd DIE ALIGN FWD/BWD SN ALARM
; L195
LOAD      M00667	// L_3rd DIE ALIGN FWD/BWD SN ALARM
AND NOT   M00008	// LEFT RESET SW PLS
OR        T0390	// L_3rd DIE ALIGN FWD/BWD SN ALARM
OUT       M00667	// L_3rd DIE ALIGN FWD/BWD SN ALARM
; L197
LOAD      P00043	// L_3rd DIE FPCB ALIGN FORWARD
OR        P00123	// L_2nd DIE FPCB ALIGN FWD/BWD
LOAD      T1036	// L_3rd DIE FPCB ALIGN BACKWARD
OR NOT    P00123	// L_2nd DIE FPCB ALIGN FWD/BWD
AND LOAD
LOAD NOT  P00043	// L_3rd DIE FPCB ALIGN FORWARD
AND NOT   T1036	// L_3rd DIE FPCB ALIGN BACKWARD
OR LOAD
TON       T0391 400	// L_3rd DIE FPCB ALIGN FWD/BWD ALARM

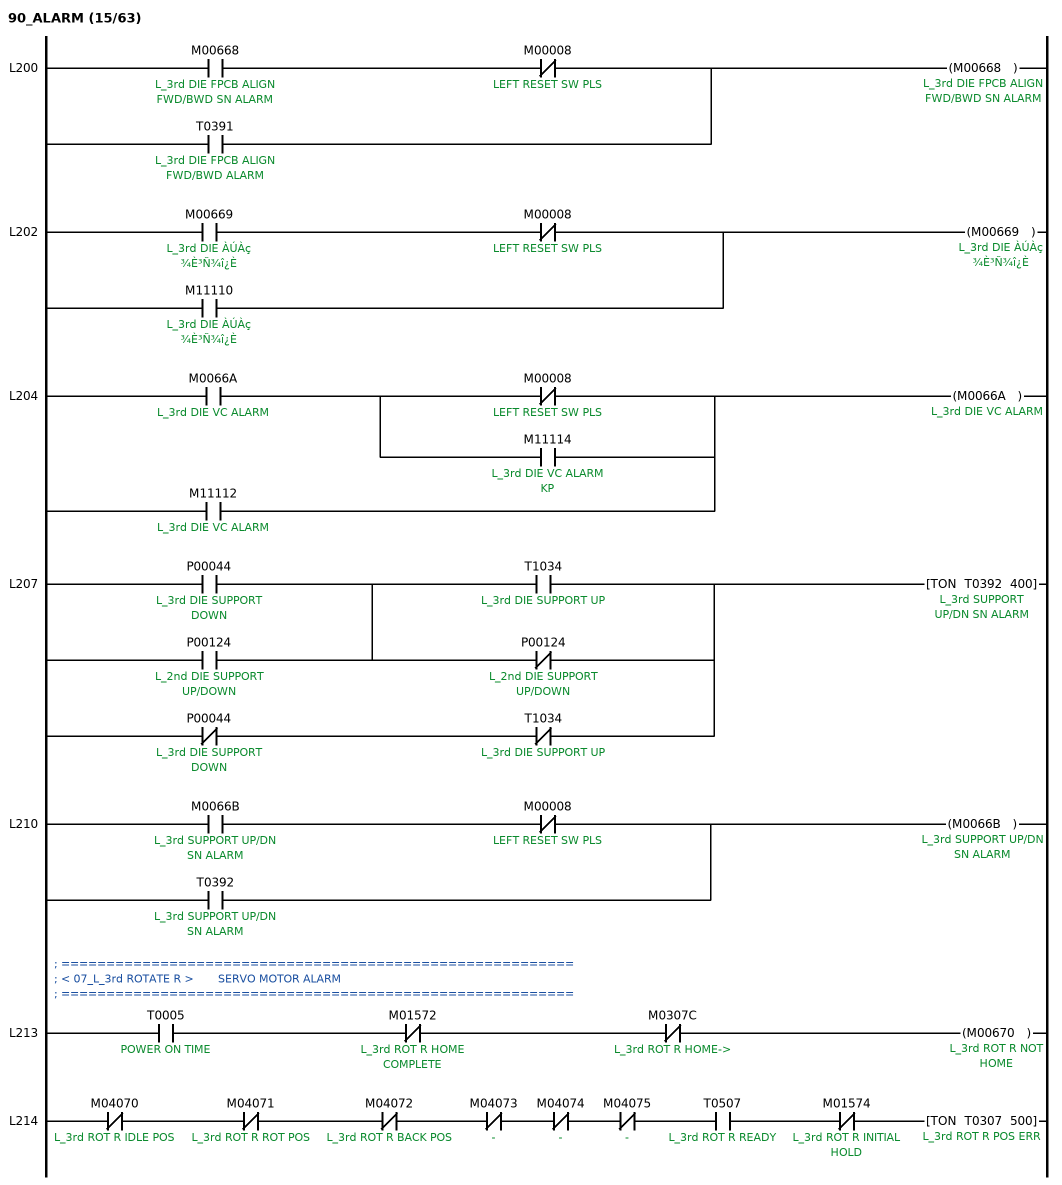
; L200
LOAD      M00668	// L_3rd DIE FPCB ALIGN FWD/BWD SN ALARM
AND NOT   M00008	// LEFT RESET SW PLS
OR        T0391	// L_3rd DIE FPCB ALIGN FWD/BWD ALARM
OUT       M00668	// L_3rd DIE FPCB ALIGN FWD/BWD SN ALARM
; L202
LOAD      M00669	// L_3rd DIE ÀÚÀç ¾È³Ñ¾î¿È
AND NOT   M00008	// LEFT RESET SW PLS
OR        M11110	// L_3rd DIE ÀÚÀç ¾È³Ñ¾î¿È
OUT       M00669	// L_3rd DIE ÀÚÀç ¾È³Ñ¾î¿È
; L204
LOAD      M0066A	// L_3rd DIE VC ALARM
LOAD NOT  M00008	// LEFT RESET SW PLS
OR        M11114	// L_3rd DIE VC ALARM KP
AND LOAD
OR        M11112	// L_3rd DIE VC ALARM
OUT       M0066A	// L_3rd DIE VC ALARM
; L207
LOAD      P00044	// L_3rd DIE SUPPORT DOWN
OR        P00124	// L_2nd DIE SUPPORT UP/DOWN
LOAD      T1034	// L_3rd DIE SUPPORT UP
OR NOT    P00124	// L_2nd DIE SUPPORT UP/DOWN
AND LOAD
LOAD NOT  P00044	// L_3rd DIE SUPPORT DOWN
AND NOT   T1034	// L_3rd DIE SUPPORT UP
OR LOAD
TON       T0392 400	// L_3rd SUPPORT UP/DN SN ALARM
; L210
LOAD      M0066B	// L_3rd SUPPORT UP/DN SN ALARM
AND NOT   M00008	// LEFT RESET SW PLS
OR        T0392	// L_3rd SUPPORT UP/DN SN ALARM
OUT       M0066B	// L_3rd SUPPORT UP/DN SN ALARM
// =========================================================
// 
//        < 07_L_3rd ROTATE R >       SERVO MOTOR ALARM
// 
// =========================================================
; L213
LOAD      T0005	// POWER ON TIME
AND NOT   M01572	// L_3rd ROT R HOME COMPLETE
AND NOT   M0307C	// L_3rd ROT R HOME->
OUT       M00670	// L_3rd ROT R NOT HOME
; L214
LOAD NOT  M04070	// L_3rd ROT R IDLE POS
AND NOT   M04071	// L_3rd ROT R ROT POS
AND NOT   M04072	// L_3rd ROT R BACK POS
AND NOT   M04073	// -
AND NOT   M04074	// -
AND NOT   M04075	// -
AND       T0507	// L_3rd ROT R READY
AND NOT   M01574	// L_3rd ROT R INITIAL HOLD
TON       T0307 500	// L_3rd ROT R POS ERR

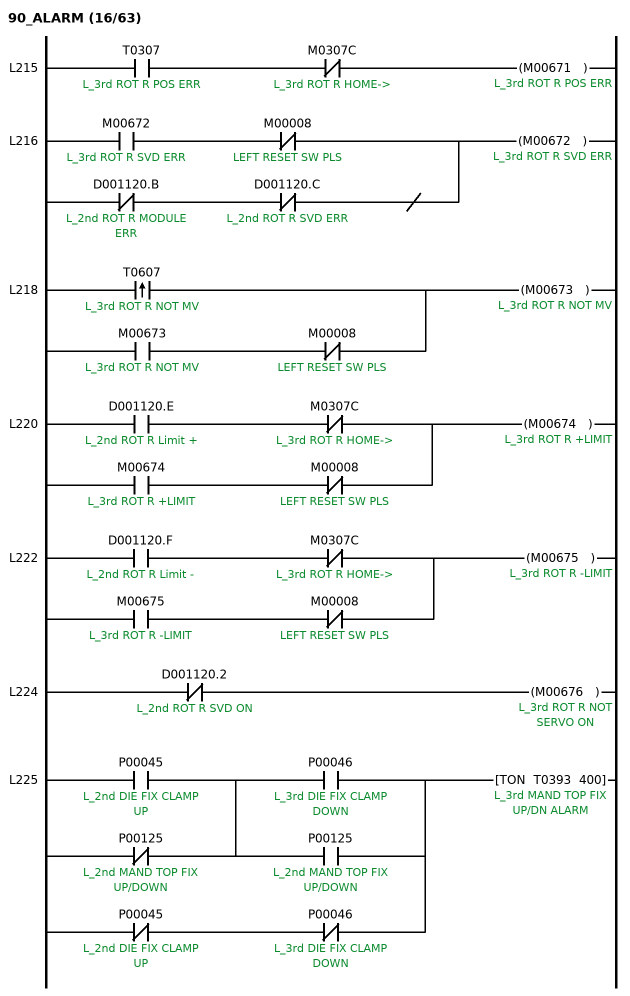
; L215
LOAD      T0307	// L_3rd ROT R POS ERR
AND NOT   M0307C	// L_3rd ROT R HOME->
OUT       M00671	// L_3rd ROT R POS ERR
; L216
LOAD      M00672	// L_3rd ROT R SVD ERR
AND NOT   M00008	// LEFT RESET SW PLS
LOAD NOT  D001120.B	// L_2nd ROT R MODULE ERR
AND NOT   D001120.C	// L_2nd ROT R SVD ERR
NOT
OR LOAD
OUT       M00672	// L_3rd ROT R SVD ERR
; L218
LOADP     T0607	// L_3rd ROT R NOT MV
LOAD      M00673	// L_3rd ROT R NOT MV
AND NOT   M00008	// LEFT RESET SW PLS
OR LOAD
OUT       M00673	// L_3rd ROT R NOT MV
; L220
LOAD      D001120.E	// L_2nd ROT R Limit +
AND NOT   M0307C	// L_3rd ROT R HOME->
LOAD      M00674	// L_3rd ROT R +LIMIT
AND NOT   M00008	// LEFT RESET SW PLS
OR LOAD
OUT       M00674	// L_3rd ROT R +LIMIT
; L222
LOAD      D001120.F	// L_2nd ROT R Limit -
AND NOT   M0307C	// L_3rd ROT R HOME->
LOAD      M00675	// L_3rd ROT R -LIMIT
AND NOT   M00008	// LEFT RESET SW PLS
OR LOAD
OUT       M00675	// L_3rd ROT R -LIMIT
; L224
LOAD NOT  D001120.2	// L_2nd ROT R SVD ON
OUT       M00676	// L_3rd ROT R NOT SERVO ON
; L225
LOAD      P00045	// L_2nd DIE FIX CLAMP UP
OR NOT    P00125	// L_2nd MAND TOP FIX UP/DOWN
LOAD      P00046	// L_3rd DIE FIX CLAMP DOWN
OR        P00125	// L_2nd MAND TOP FIX UP/DOWN
AND LOAD
LOAD NOT  P00045	// L_2nd DIE FIX CLAMP UP
AND NOT   P00046	// L_3rd DIE FIX CLAMP DOWN
OR LOAD
TON       T0393 400	// L_3rd MAND TOP FIX UP/DN ALARM

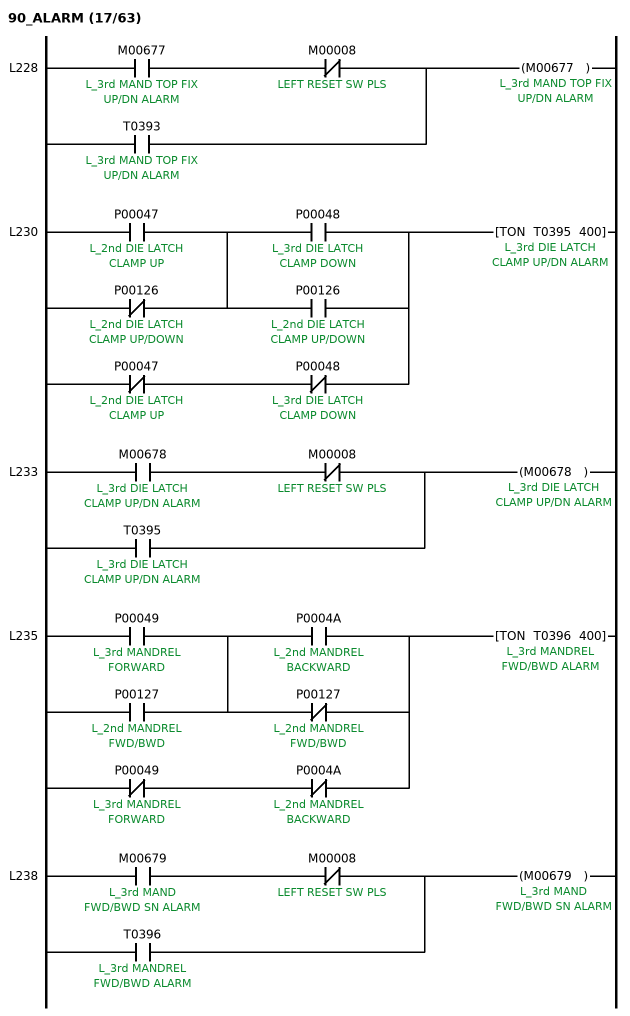
; L228
LOAD      M00677	// L_3rd MAND TOP FIX UP/DN ALARM
AND NOT   M00008	// LEFT RESET SW PLS
OR        T0393	// L_3rd MAND TOP FIX UP/DN ALARM
OUT       M00677	// L_3rd MAND TOP FIX UP/DN ALARM
; L230
LOAD      P00047	// L_2nd DIE LATCH CLAMP UP
OR NOT    P00126	// L_2nd DIE LATCH CLAMP UP/DOWN
LOAD      P00048	// L_3rd DIE LATCH CLAMP DOWN
OR        P00126	// L_2nd DIE LATCH CLAMP UP/DOWN
AND LOAD
LOAD NOT  P00047	// L_2nd DIE LATCH CLAMP UP
AND NOT   P00048	// L_3rd DIE LATCH CLAMP DOWN
OR LOAD
TON       T0395 400	// L_3rd DIE LATCH CLAMP UP/DN ALARM
; L233
LOAD      M00678	// L_3rd DIE LATCH CLAMP UP/DN ALARM
AND NOT   M00008	// LEFT RESET SW PLS
OR        T0395	// L_3rd DIE LATCH CLAMP UP/DN ALARM
OUT       M00678	// L_3rd DIE LATCH CLAMP UP/DN ALARM
; L235
LOAD      P00049	// L_3rd MANDREL FORWARD
OR        P00127	// L_2nd MANDREL FWD/BWD
LOAD      P0004A	// L_2nd MANDREL BACKWARD
OR NOT    P00127	// L_2nd MANDREL FWD/BWD
AND LOAD
LOAD NOT  P00049	// L_3rd MANDREL FORWARD
AND NOT   P0004A	// L_2nd MANDREL BACKWARD
OR LOAD
TON       T0396 400	// L_3rd MANDREL FWD/BWD ALARM
; L238
LOAD      M00679	// L_3rd MAND FWD/BWD SN ALARM
AND NOT   M00008	// LEFT RESET SW PLS
OR        T0396	// L_3rd MANDREL FWD/BWD ALARM
OUT       M00679	// L_3rd MAND FWD/BWD SN ALARM

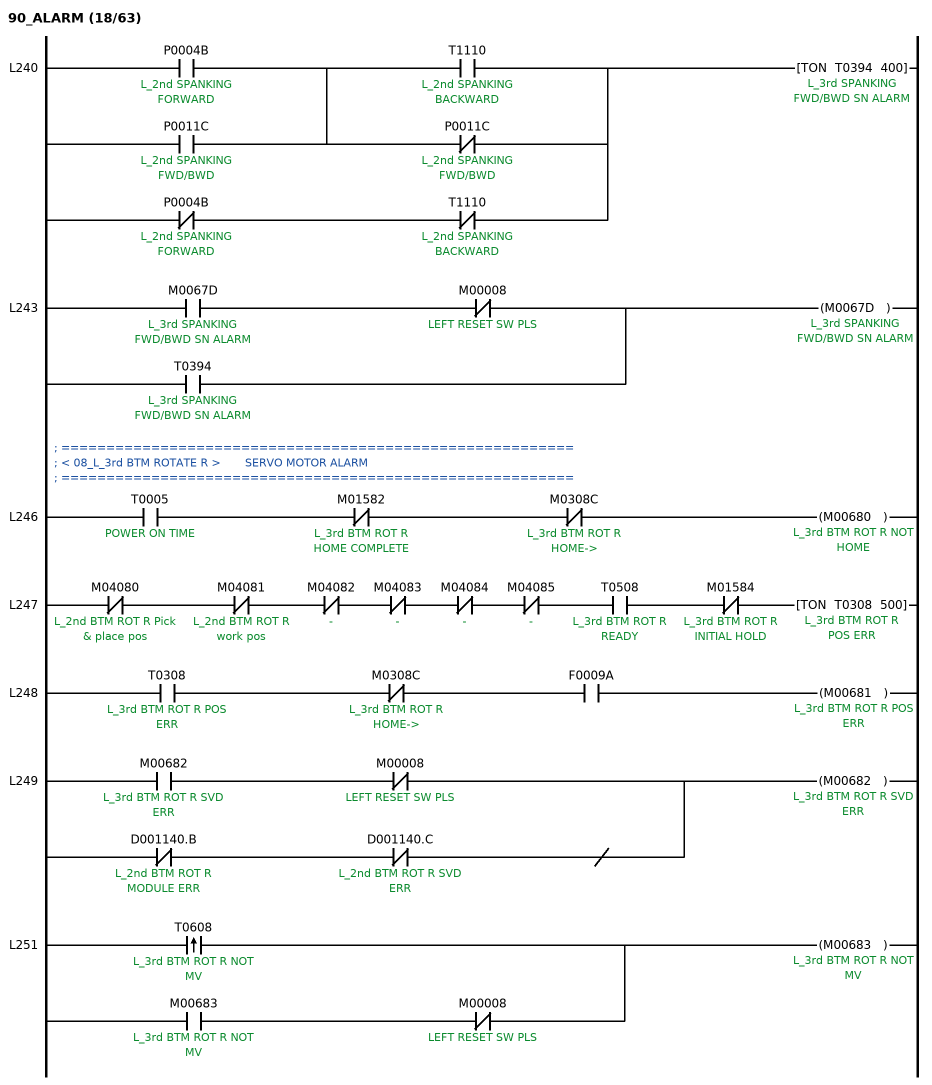
; L240
LOAD      P0004B	// L_2nd SPANKING FORWARD
OR        P0011C	// L_2nd SPANKING FWD/BWD
LOAD      T1110	// L_2nd SPANKING BACKWARD
OR NOT    P0011C	// L_2nd SPANKING FWD/BWD
AND LOAD
LOAD NOT  P0004B	// L_2nd SPANKING FORWARD
AND NOT   T1110	// L_2nd SPANKING BACKWARD
OR LOAD
TON       T0394 400	// L_3rd SPANKING FWD/BWD SN ALARM
; L243
LOAD      M0067D	// L_3rd SPANKING FWD/BWD SN ALARM
AND NOT   M00008	// LEFT RESET SW PLS
OR        T0394	// L_3rd SPANKING FWD/BWD SN ALARM
OUT       M0067D	// L_3rd SPANKING FWD/BWD SN ALARM
// =========================================================
// 
//        < 08_L_3rd BTM ROTATE R >       SERVO MOTOR ALARM
// 
// =========================================================
; L246
LOAD      T0005	// POWER ON TIME
AND NOT   M01582	// L_3rd BTM ROT R HOME COMPLETE
AND NOT   M0308C	// L_3rd BTM ROT R HOME->
OUT       M00680	// L_3rd BTM ROT R NOT HOME
; L247
LOAD NOT  M04080	// L_2nd BTM ROT R Pick & place pos
AND NOT   M04081	// L_2nd BTM ROT R work pos
AND NOT   M04082	// -
AND NOT   M04083	// -
AND NOT   M04084	// -
AND NOT   M04085	// -
AND       T0508	// L_3rd BTM ROT R READY
AND NOT   M01584	// L_3rd BTM ROT R INITIAL HOLD
TON       T0308 500	// L_3rd BTM ROT R POS ERR
; L248
LOAD      T0308	// L_3rd BTM ROT R POS ERR
AND NOT   M0308C	// L_3rd BTM ROT R HOME->
AND       F0009A
OUT       M00681	// L_3rd BTM ROT R POS ERR
; L249
LOAD      M00682	// L_3rd BTM ROT R SVD ERR
AND NOT   M00008	// LEFT RESET SW PLS
LOAD NOT  D001140.B	// L_2nd BTM ROT R MODULE ERR
AND NOT   D001140.C	// L_2nd BTM ROT R SVD ERR
NOT
OR LOAD
OUT       M00682	// L_3rd BTM ROT R SVD ERR
; L251
LOADP     T0608	// L_3rd BTM ROT R NOT MV
LOAD      M00683	// L_3rd BTM ROT R NOT MV
AND NOT   M00008	// LEFT RESET SW PLS
OR LOAD
OUT       M00683	// L_3rd BTM ROT R NOT MV

